  STRUCT
   S711A_WELD_DATA : STRUCT
    STATION_MAIN : WORD ;
    DISTINCTION_LH_RH : WORD ;
    STAION_NUMBER : WORD ;
    VIN_NUMBER1 : WORD ;
    VIN_NUMBER2 : WORD ;
    VIN_NUMBER3 : WORD ;
    VIN_NUMBER4 : WORD ;
    SEQ_NUMBER1 : WORD ;
    SEQ_NUMBER2 : WORD ;
    RBT1_BT_CODE_NO : WORD ;
    RBT1_WELD_COUNT : WORD ;
    RBT2_BT_CODE_NO : WORD ;
    RBT2_WELD_COUNT : WORD ;
    RBT3_BT_CODE_NO : WORD ;
    RBT3_WELD_COUNT : WORD ;
    RBT4_BT_CODE_NO : WORD ;
    RBT4_WELD_COUNT : WORD ;
    RBT5_BT_CODE_NO : WORD ;
    RBT5_WELD_COUNT : WORD ;
    RBT6_BT_CODE_NO : WORD ;
    RBT6_WELD_COUNT : WORD ;
    RBT7_BT_CODE_NO : WORD ;
    RBT7_WELD_COUNT : WORD ;
    RBT8_BT_CODE_NO : WORD ;
    RBT8_WELD_COUNT : WORD ;
    RBT9_BT_CODE_NO : WORD ;
    RBT9_WELD_COUNT : WORD ;
    RBT10_BT_CODE_NO : WORD ;
    RBT10_WELD_COUNT : WORD ;
    RBT11_BT_CODE_NO : WORD ;
    RBT11_WELD_COUNT : WORD ;
    RBT12_BT_CODE_NO : WORD ;
    RBT12_WELD_COUNT : WORD ;
    RBT13_BT_CODE_NO : WORD ;
    RBT13_WELD_COUNT : WORD ;
    RBT14_BT_CODE_NO : WORD ;
    RBT14_WELD_COUNT : WORD ;
    RBT15_BT_CODE_NO : WORD ;
    RBT15_WELD_COUNT : WORD ;
    RBT16_BT_CODE_NO : WORD ;
    RBT16_WELD_COUNT : WORD ;
    RBT17_BT_CODE_NO : WORD ;
    RBT17_WELD_COUNT : WORD ;
    RBT18_BT_CODE_NO : WORD ;
    RBT18_WELD_COUNT : WORD ;
    RBT19_BT_CODE_NO : WORD ;
    RBT19_WELD_COUNT : WORD ;
    RBT20_BT_CODE_NO : WORD ;
    RBT20_WELD_COUNT : WORD ;
    RBT21_BT_CODE_NO : WORD ;
    RBT21_WELD_COUNT : WORD ;
    RBT22_BT_CODE_NO : WORD ;
    RBT22_WELD_COUNT : WORD ;
    RBT23_BT_CODE_NO : WORD ;
    RBT23_WELD_COUNT : WORD ;
    RBT24_BT_CODE_NO : WORD ;
    RBT24_WELD_COUNT : WORD ;
    WELD_DETERMINES_RESULT : WORD ;
    WELD_CHECK_SUM : WORD ;
    SPARE1 : WORD ;
    SPARE2 : WORD ;
    SPARE3 : WORD ;
    SPARE4 : WORD ;
    SPARE5 : WORD ;
    SPARE6 : WORD ;
    SPARE7 : WORD ;
    SPARE8 : WORD ;
    SPARE9 : WORD ;
    SPARE10 : WORD ;
    SPARE11 : WORD ;
    SPARE12 : WORD ;
    SPARE13 : WORD ;
    SPARE14 : WORD ;
    SPARE15 : WORD ;
    SPARE16 : WORD ;
    SPARE17 : WORD ;
    SPARE18 : WORD ;
    SPARE19 : WORD ;
    SPARE20 : WORD ;
    SPARE21 : WORD ;
    SPARE22 : WORD ;
    SPARE23 : WORD ;
    SPARE24 : WORD ;
    SPARE25 : WORD ;
    SPARE26 : WORD ;
    SPARE27 : WORD ;
    SPARE28 : WORD ;
    SPARE29 : WORD ;
    SPARE30 : WORD ;
    SPARE31 : WORD ;
    RBT1_WELD_COUNT_OK : BOOL ;
    RBT1_WELD_COUNT_NG : BOOL ;
    RBT1_PASS_T_TAG : BOOL ;
    RBT1_PASS_L_TAG : BOOL ;
    RBT2_WELD_COUNT_OK : BOOL ;
    RBT2_WELD_COUNT_NG : BOOL ;
    RBT2_PASS_T_TAG : BOOL ;
    RBT2_PASS_L_TAG : BOOL ;
    RBT3_WELD_COUNT_OK : BOOL ;
    RBT3_WELD_COUNT_NG : BOOL ;
    RBT3_PASS_T_TAG : BOOL ;
    RBT3_PASS_L_TAG : BOOL ;
    RBT4_WELD_COUNT_OK : BOOL ;
    RBT4_WELD_COUNT_NG : BOOL ;
    RBT4_PASS_T_TAG : BOOL ;
    RBT4_PASS_L_TAG : BOOL ;
    RBT5_WELD_COUNT_OK : BOOL ;
    RBT5_WELD_COUNT_NG : BOOL ;
    RBT5_PASS_T_TAG : BOOL ;
    RBT5_PASS_L_TAG : BOOL ;
    RBT6_WELD_COUNT_OK : BOOL ;
    RBT6_WELD_COUNT_NG : BOOL ;
    RBT6_PASS_T_TAG : BOOL ;
    RBT6_PASS_L_TAG : BOOL ;
    RBT7_WELD_COUNT_OK : BOOL ;
    RBT7_WELD_COUNT_NG : BOOL ;
    RBT7_PASS_T_TAG : BOOL ;
    RBT7_PASS_L_TAG : BOOL ;
    RBT8_WELD_COUNT_OK : BOOL ;
    RBT8_WELD_COUNT_NG : BOOL ;
    RBT8_PASS_T_TAG : BOOL ;
    RBT8_PASS_L_TAG : BOOL ;
    RBT9_WELD_COUNT_OK : BOOL ;
    RBT9_WELD_COUNT_NG : BOOL ;
    RBT9_PASS_T_TAG : BOOL ;
    RBT9_PASS_L_TAG : BOOL ;
    RBT10_WELD_COUNT_OK : BOOL ;
    RBT10_WELD_COUNT_NG : BOOL ;
    RBT10_PASS_T_TAG : BOOL ;
    RBT10_PASS_L_TAG : BOOL ;
    RBT11_WELD_COUNT_OK : BOOL ;
    RBT11_WELD_COUNT_NG : BOOL ;
    RBT11_PASS_T_TAG : BOOL ;
    RBT11_PASS_L_TAG : BOOL ;
    RBT12_WELD_COUNT_OK : BOOL ;
    RBT12_WELD_COUNT_NG : BOOL ;
    RBT12_PASS_T_TAG : BOOL ;
    RBT12_PASS_L_TAG : BOOL ;
    RBT13_WELD_COUNT_OK : BOOL ;
    RBT13_WELD_COUNT_NG : BOOL ;
    RBT13_PASS_T_TAG : BOOL ;
    RBT13_PASS_L_TAG : BOOL ;
    RBT14_WELD_COUNT_OK : BOOL ;
    RBT14_WELD_COUNT_NG : BOOL ;
    RBT14_PASS_T_TAG : BOOL ;
    RBT14_PASS_L_TAG : BOOL ;
    RBT15_WELD_COUNT_OK : BOOL ;
    RBT15_WELD_COUNT_NG : BOOL ;
    RBT15_PASS_T_TAG : BOOL ;
    RBT15_PASS_L_TAG : BOOL ;
    RBT16_WELD_COUNT_OK : BOOL ;
    RBT16_WELD_COUNT_NG : BOOL ;
    RBT16_PASS_T_TAG : BOOL ;
    RBT16_PASS_L_TAG : BOOL ;
    RBT17_WELD_COUNT_OK : BOOL ;
    RBT17_WELD_COUNT_NG : BOOL ;
    RBT17_PASS_T_TAG : BOOL ;
    RBT17_PASS_L_TAG : BOOL ;
    RBT18_WELD_COUNT_OK : BOOL ;
    RBT18_WELD_COUNT_NG : BOOL ;
    RBT18_PASS_T_TAG : BOOL ;
    RBT18_PASS_L_TAG : BOOL ;
    RBT19_WELD_COUNT_OK : BOOL ;
    RBT19_WELD_COUNT_NG : BOOL ;
    RBT19_PASS_T_TAG : BOOL ;
    RBT19_PASS_L_TAG : BOOL ;
    RBT20_WELD_COUNT_OK : BOOL ;
    RBT20_WELD_COUNT_NG : BOOL ;
    RBT20_PASS_T_TAG : BOOL ;
    RBT20_PASS_L_TAG : BOOL ;
    RBT21_WELD_COUNT_OK : BOOL ;
    RBT21_WELD_COUNT_NG : BOOL ;
    RBT21_PASS_T_TAG : BOOL ;
    RBT21_PASS_L_TAG : BOOL ;
    RBT22_WELD_COUNT_OK : BOOL ;
    RBT22_WELD_COUNT_NG : BOOL ;
    RBT22_PASS_T_TAG : BOOL ;
    RBT22_PASS_L_TAG : BOOL ;
    RBT23_WELD_COUNT_OK : BOOL ;
    RBT23_WELD_COUNT_NG : BOOL ;
    RBT23_PASS_T_TAG : BOOL ;
    RBT23_PASS_L_TAG : BOOL ;
    RBT24_WELD_COUNT_OK : BOOL ;
    RBT24_WELD_COUNT_NG : BOOL ;
    RBT24_PASS_T_TAG : BOOL ;
    RBT24_PASS_L_TAG : BOOL ;
    SPARE100 : BOOL ;
    SPARE101 : BOOL ;
    SPARE102 : BOOL ;
    SPARE103 : BOOL ;
    SPARE104 : BOOL ;
    SPARE105 : BOOL ;
    SPARE106 : BOOL ;
    SPARE107 : BOOL ;
    SPARE108 : BOOL ;
    SPARE109 : BOOL ;
    SPARE110 : BOOL ;
    SPARE111 : BOOL ;
    SPARE112 : BOOL ;
    SPARE113 : BOOL ;
    SPARE114 : BOOL ;
    SPARE115 : BOOL ;
    SPARE116 : WORD ;
    SPARE117 : WORD ;
    SPARE118 : WORD ;
   END_STRUCT ;
   S706_WELD_DATA : STRUCT
    STATION_MAIN : WORD ;
    DISTINCTION_LH_RH : WORD ;
    STAION_NUMBER : WORD ;
    VIN_NUMBER1 : WORD ;
    VIN_NUMBER2 : WORD ;
    VIN_NUMBER3 : WORD ;
    VIN_NUMBER4 : WORD ;
    SEQ_NUMBER1 : WORD ;
    SEQ_NUMBER2 : WORD ;
    RBT1_BT_CODE_NO : WORD ;
    RBT1_WELD_COUNT : WORD ;
    RBT2_BT_CODE_NO : WORD ;
    RBT2_WELD_COUNT : WORD ;
    RBT3_BT_CODE_NO : WORD ;
    RBT3_WELD_COUNT : WORD ;
    RBT4_BT_CODE_NO : WORD ;
    RBT4_WELD_COUNT : WORD ;
    RBT5_BT_CODE_NO : WORD ;
    RBT5_WELD_COUNT : WORD ;
    RBT6_BT_CODE_NO : WORD ;
    RBT6_WELD_COUNT : WORD ;
    RBT7_BT_CODE_NO : WORD ;
    RBT7_WELD_COUNT : WORD ;
    RBT8_BT_CODE_NO : WORD ;
    RBT8_WELD_COUNT : WORD ;
    RBT9_BT_CODE_NO : WORD ;
    RBT9_WELD_COUNT : WORD ;
    RBT10_BT_CODE_NO : WORD ;
    RBT10_WELD_COUNT : WORD ;
    RBT11_BT_CODE_NO : WORD ;
    RBT11_WELD_COUNT : WORD ;
    RBT12_BT_CODE_NO : WORD ;
    RBT12_WELD_COUNT : WORD ;
    RBT13_BT_CODE_NO : WORD ;
    RBT13_WELD_COUNT : WORD ;
    RBT14_BT_CODE_NO : WORD ;
    RBT14_WELD_COUNT : WORD ;
    RBT15_BT_CODE_NO : WORD ;
    RBT15_WELD_COUNT : WORD ;
    RBT16_BT_CODE_NO : WORD ;
    RBT16_WELD_COUNT : WORD ;
    RBT17_BT_CODE_NO : WORD ;
    RBT17_WELD_COUNT : WORD ;
    RBT18_BT_CODE_NO : WORD ;
    RBT18_WELD_COUNT : WORD ;
    RBT19_BT_CODE_NO : WORD ;
    RBT19_WELD_COUNT : WORD ;
    RBT20_BT_CODE_NO : WORD ;
    RBT20_WELD_COUNT : WORD ;
    RBT21_BT_CODE_NO : WORD ;
    RBT21_WELD_COUNT : WORD ;
    RBT22_BT_CODE_NO : WORD ;
    RBT22_WELD_COUNT : WORD ;
    RBT23_BT_CODE_NO : WORD ;
    RBT23_WELD_COUNT : WORD ;
    RBT24_BT_CODE_NO : WORD ;
    RBT24_WELD_COUNT : WORD ;
    WELD_DETERMINES_RESULT : WORD ;
    WELD_CHECK_SUM : WORD ;
    SPARE1 : WORD ;
    SPARE2 : WORD ;
    SPARE3 : WORD ;
    SPARE4 : WORD ;
    SPARE5 : WORD ;
    SPARE6 : WORD ;
    SPARE7 : WORD ;
    SPARE8 : WORD ;
    SPARE9 : WORD ;
    SPARE10 : WORD ;
    SPARE11 : WORD ;
    SPARE12 : WORD ;
    SPARE13 : WORD ;
    SPARE14 : WORD ;
    SPARE15 : WORD ;
    SPARE16 : WORD ;
    SPARE17 : WORD ;
    SPARE18 : WORD ;
    SPARE19 : WORD ;
    SPARE20 : WORD ;
    SPARE21 : WORD ;
    SPARE22 : WORD ;
    SPARE23 : WORD ;
    SPARE24 : WORD ;
    SPARE25 : WORD ;
    SPARE26 : WORD ;
    SPARE27 : WORD ;
    SPARE28 : WORD ;
    SPARE29 : WORD ;
    SPARE30 : WORD ;
    SPARE31 : WORD ;
    RBT1_WELD_COUNT_OK : BOOL ;
    RBT1_WELD_COUNT_NG : BOOL ;
    RBT1_PASS_T_TAG : BOOL ;
    RBT1_PASS_L_TAG : BOOL ;
    RBT2_WELD_COUNT_OK : BOOL ;
    RBT2_WELD_COUNT_NG : BOOL ;
    RBT2_PASS_T_TAG : BOOL ;
    RBT2_PASS_L_TAG : BOOL ;
    RBT3_WELD_COUNT_OK : BOOL ;
    RBT3_WELD_COUNT_NG : BOOL ;
    RBT3_PASS_T_TAG : BOOL ;
    RBT3_PASS_L_TAG : BOOL ;
    RBT4_WELD_COUNT_OK : BOOL ;
    RBT4_WELD_COUNT_NG : BOOL ;
    RBT4_PASS_T_TAG : BOOL ;
    RBT4_PASS_L_TAG : BOOL ;
    RBT5_WELD_COUNT_OK : BOOL ;
    RBT5_WELD_COUNT_NG : BOOL ;
    RBT5_PASS_T_TAG : BOOL ;
    RBT5_PASS_L_TAG : BOOL ;
    RBT6_WELD_COUNT_OK : BOOL ;
    RBT6_WELD_COUNT_NG : BOOL ;
    RBT6_PASS_T_TAG : BOOL ;
    RBT6_PASS_L_TAG : BOOL ;
    RBT7_WELD_COUNT_OK : BOOL ;
    RBT7_WELD_COUNT_NG : BOOL ;
    RBT7_PASS_T_TAG : BOOL ;
    RBT7_PASS_L_TAG : BOOL ;
    RBT8_WELD_COUNT_OK : BOOL ;
    RBT8_WELD_COUNT_NG : BOOL ;
    RBT8_PASS_T_TAG : BOOL ;
    RBT8_PASS_L_TAG : BOOL ;
    RBT9_WELD_COUNT_OK : BOOL ;
    RBT9_WELD_COUNT_NG : BOOL ;
    RBT9_PASS_T_TAG : BOOL ;
    RBT9_PASS_L_TAG : BOOL ;
    RBT10_WELD_COUNT_OK : BOOL ;
    RBT10_WELD_COUNT_NG : BOOL ;
    RBT10_PASS_T_TAG : BOOL ;
    RBT10_PASS_L_TAG : BOOL ;
    RBT11_WELD_COUNT_OK : BOOL ;
    RBT11_WELD_COUNT_NG : BOOL ;
    RBT11_PASS_T_TAG : BOOL ;
    RBT11_PASS_L_TAG : BOOL ;
    RBT12_WELD_COUNT_OK : BOOL ;
    RBT12_WELD_COUNT_NG : BOOL ;
    RBT12_PASS_T_TAG : BOOL ;
    RBT12_PASS_L_TAG : BOOL ;
    RBT13_WELD_COUNT_OK : BOOL ;
    RBT13_WELD_COUNT_NG : BOOL ;
    RBT13_PASS_T_TAG : BOOL ;
    RBT13_PASS_L_TAG : BOOL ;
    RBT14_WELD_COUNT_OK : BOOL ;
    RBT14_WELD_COUNT_NG : BOOL ;
    RBT14_PASS_T_TAG : BOOL ;
    RBT14_PASS_L_TAG : BOOL ;
    RBT15_WELD_COUNT_OK : BOOL ;
    RBT15_WELD_COUNT_NG : BOOL ;
    RBT15_PASS_T_TAG : BOOL ;
    RBT15_PASS_L_TAG : BOOL ;
    RBT16_WELD_COUNT_OK : BOOL ;
    RBT16_WELD_COUNT_NG : BOOL ;
    RBT16_PASS_T_TAG : BOOL ;
    RBT16_PASS_L_TAG : BOOL ;
    RBT17_WELD_COUNT_OK : BOOL ;
    RBT17_WELD_COUNT_NG : BOOL ;
    RBT17_PASS_T_TAG : BOOL ;
    RBT17_PASS_L_TAG : BOOL ;
    RBT18_WELD_COUNT_OK : BOOL ;
    RBT18_WELD_COUNT_NG : BOOL ;
    RBT18_PASS_T_TAG : BOOL ;
    RBT18_PASS_L_TAG : BOOL ;
    RBT19_WELD_COUNT_OK : BOOL ;
    RBT19_WELD_COUNT_NG : BOOL ;
    RBT19_PASS_T_TAG : BOOL ;
    RBT19_PASS_L_TAG : BOOL ;
    RBT20_WELD_COUNT_OK : BOOL ;
    RBT20_WELD_COUNT_NG : BOOL ;
    RBT20_PASS_T_TAG : BOOL ;
    RBT20_PASS_L_TAG : BOOL ;
    RBT21_WELD_COUNT_OK : BOOL ;
    RBT21_WELD_COUNT_NG : BOOL ;
    RBT21_PASS_T_TAG : BOOL ;
    RBT21_PASS_L_TAG : BOOL ;
    RBT22_WELD_COUNT_OK : BOOL ;
    RBT22_WELD_COUNT_NG : BOOL ;
    RBT22_PASS_T_TAG : BOOL ;
    RBT22_PASS_L_TAG : BOOL ;
    RBT23_WELD_COUNT_OK : BOOL ;
    RBT23_WELD_COUNT_NG : BOOL ;
    RBT23_PASS_T_TAG : BOOL ;
    RBT23_PASS_L_TAG : BOOL ;
    RBT24_WELD_COUNT_OK : BOOL ;
    RBT24_WELD_COUNT_NG : BOOL ;
    RBT24_PASS_T_TAG : BOOL ;
    RBT24_PASS_L_TAG : BOOL ;
    SPARE100 : BOOL ;
    SPARE101 : BOOL ;
    SPARE102 : BOOL ;
    SPARE103 : BOOL ;
    SPARE104 : BOOL ;
    SPARE105 : BOOL ;
    SPARE106 : BOOL ;
    SPARE107 : BOOL ;
    SPARE108 : BOOL ;
    SPARE109 : BOOL ;
    SPARE110 : BOOL ;
    SPARE111 : BOOL ;
    SPARE112 : BOOL ;
    SPARE113 : BOOL ;
    SPARE114 : BOOL ;
    SPARE115 : BOOL ;
    SPARE116 : WORD ;
    SPARE117 : WORD ;
    SPARE118 : WORD ;
   END_STRUCT ;
   S711_WELD_DATA : STRUCT
    STATION_MAIN : WORD ;
    DISTINCTION_LH_RH : WORD ;
    STAION_NUMBER : WORD ;
    VIN_NUMBER1 : WORD ;
    VIN_NUMBER2 : WORD ;
    VIN_NUMBER3 : WORD ;
    VIN_NUMBER4 : WORD ;
    SEQ_NUMBER1 : WORD ;
    SEQ_NUMBER2 : WORD ;
    RBT1_BT_CODE_NO : WORD ;
    RBT1_WELD_COUNT : WORD ;
    RBT2_BT_CODE_NO : WORD ;
    RBT2_WELD_COUNT : WORD ;
    RBT3_BT_CODE_NO : WORD ;
    RBT3_WELD_COUNT : WORD ;
    RBT4_BT_CODE_NO : WORD ;
    RBT4_WELD_COUNT : WORD ;
    RBT5_BT_CODE_NO : WORD ;
    RBT5_WELD_COUNT : WORD ;
    RBT6_BT_CODE_NO : WORD ;
    RBT6_WELD_COUNT : WORD ;
    RBT7_BT_CODE_NO : WORD ;
    RBT7_WELD_COUNT : WORD ;
    RBT8_BT_CODE_NO : WORD ;
    RBT8_WELD_COUNT : WORD ;
    RBT9_BT_CODE_NO : WORD ;
    RBT9_WELD_COUNT : WORD ;
    RBT10_BT_CODE_NO : WORD ;
    RBT10_WELD_COUNT : WORD ;
    RBT11_BT_CODE_NO : WORD ;
    RBT11_WELD_COUNT : WORD ;
    RBT12_BT_CODE_NO : WORD ;
    RBT12_WELD_COUNT : WORD ;
    RBT13_BT_CODE_NO : WORD ;
    RBT13_WELD_COUNT : WORD ;
    RBT14_BT_CODE_NO : WORD ;
    RBT14_WELD_COUNT : WORD ;
    RBT15_BT_CODE_NO : WORD ;
    RBT15_WELD_COUNT : WORD ;
    RBT16_BT_CODE_NO : WORD ;
    RBT16_WELD_COUNT : WORD ;
    RBT17_BT_CODE_NO : WORD ;
    RBT17_WELD_COUNT : WORD ;
    RBT18_BT_CODE_NO : WORD ;
    RBT18_WELD_COUNT : WORD ;
    RBT19_BT_CODE_NO : WORD ;
    RBT19_WELD_COUNT : WORD ;
    RBT20_BT_CODE_NO : WORD ;
    RBT20_WELD_COUNT : WORD ;
    RBT21_BT_CODE_NO : WORD ;
    RBT21_WELD_COUNT : WORD ;
    RBT22_BT_CODE_NO : WORD ;
    RBT22_WELD_COUNT : WORD ;
    RBT23_BT_CODE_NO : WORD ;
    RBT23_WELD_COUNT : WORD ;
    RBT24_BT_CODE_NO : WORD ;
    RBT24_WELD_COUNT : WORD ;
    WELD_DETERMINES_RESULT : WORD ;
    WELD_CHECK_SUM : WORD ;
    SPARE1 : WORD ;
    SPARE2 : WORD ;
    SPARE3 : WORD ;
    SPARE4 : WORD ;
    SPARE5 : WORD ;
    SPARE6 : WORD ;
    SPARE7 : WORD ;
    SPARE8 : WORD ;
    SPARE9 : WORD ;
    SPARE10 : WORD ;
    SPARE11 : WORD ;
    SPARE12 : WORD ;
    SPARE13 : WORD ;
    SPARE14 : WORD ;
    SPARE15 : WORD ;
    SPARE16 : WORD ;
    SPARE17 : WORD ;
    SPARE18 : WORD ;
    SPARE19 : WORD ;
    SPARE20 : WORD ;
    SPARE21 : WORD ;
    SPARE22 : WORD ;
    SPARE23 : WORD ;
    SPARE24 : WORD ;
    SPARE25 : WORD ;
    SPARE26 : WORD ;
    SPARE27 : WORD ;
    SPARE28 : WORD ;
    SPARE29 : WORD ;
    SPARE30 : WORD ;
    SPARE31 : WORD ;
    RBT1_WELD_COUNT_OK : BOOL ;
    RBT1_WELD_COUNT_NG : BOOL ;
    RBT1_PASS_T_TAG : BOOL ;
    RBT1_PASS_L_TAG : BOOL ;
    RBT2_WELD_COUNT_OK : BOOL ;
    RBT2_WELD_COUNT_NG : BOOL ;
    RBT2_PASS_T_TAG : BOOL ;
    RBT2_PASS_L_TAG : BOOL ;
    RBT3_WELD_COUNT_OK : BOOL ;
    RBT3_WELD_COUNT_NG : BOOL ;
    RBT3_PASS_T_TAG : BOOL ;
    RBT3_PASS_L_TAG : BOOL ;
    RBT4_WELD_COUNT_OK : BOOL ;
    RBT4_WELD_COUNT_NG : BOOL ;
    RBT4_PASS_T_TAG : BOOL ;
    RBT4_PASS_L_TAG : BOOL ;
    RBT5_WELD_COUNT_OK : BOOL ;
    RBT5_WELD_COUNT_NG : BOOL ;
    RBT5_PASS_T_TAG : BOOL ;
    RBT5_PASS_L_TAG : BOOL ;
    RBT6_WELD_COUNT_OK : BOOL ;
    RBT6_WELD_COUNT_NG : BOOL ;
    RBT6_PASS_T_TAG : BOOL ;
    RBT6_PASS_L_TAG : BOOL ;
    RBT7_WELD_COUNT_OK : BOOL ;
    RBT7_WELD_COUNT_NG : BOOL ;
    RBT7_PASS_T_TAG : BOOL ;
    RBT7_PASS_L_TAG : BOOL ;
    RBT8_WELD_COUNT_OK : BOOL ;
    RBT8_WELD_COUNT_NG : BOOL ;
    RBT8_PASS_T_TAG : BOOL ;
    RBT8_PASS_L_TAG : BOOL ;
    RBT9_WELD_COUNT_OK : BOOL ;
    RBT9_WELD_COUNT_NG : BOOL ;
    RBT9_PASS_T_TAG : BOOL ;
    RBT9_PASS_L_TAG : BOOL ;
    RBT10_WELD_COUNT_OK : BOOL ;
    RBT10_WELD_COUNT_NG : BOOL ;
    RBT10_PASS_T_TAG : BOOL ;
    RBT10_PASS_L_TAG : BOOL ;
    RBT11_WELD_COUNT_OK : BOOL ;
    RBT11_WELD_COUNT_NG : BOOL ;
    RBT11_PASS_T_TAG : BOOL ;
    RBT11_PASS_L_TAG : BOOL ;
    RBT12_WELD_COUNT_OK : BOOL ;
    RBT12_WELD_COUNT_NG : BOOL ;
    RBT12_PASS_T_TAG : BOOL ;
    RBT12_PASS_L_TAG : BOOL ;
    RBT13_WELD_COUNT_OK : BOOL ;
    RBT13_WELD_COUNT_NG : BOOL ;
    RBT13_PASS_T_TAG : BOOL ;
    RBT13_PASS_L_TAG : BOOL ;
    RBT14_WELD_COUNT_OK : BOOL ;
    RBT14_WELD_COUNT_NG : BOOL ;
    RBT14_PASS_T_TAG : BOOL ;
    RBT14_PASS_L_TAG : BOOL ;
    RBT15_WELD_COUNT_OK : BOOL ;
    RBT15_WELD_COUNT_NG : BOOL ;
    RBT15_PASS_T_TAG : BOOL ;
    RBT15_PASS_L_TAG : BOOL ;
    RBT16_WELD_COUNT_OK : BOOL ;
    RBT16_WELD_COUNT_NG : BOOL ;
    RBT16_PASS_T_TAG : BOOL ;
    RBT16_PASS_L_TAG : BOOL ;
    RBT17_WELD_COUNT_OK : BOOL ;
    RBT17_WELD_COUNT_NG : BOOL ;
    RBT17_PASS_T_TAG : BOOL ;
    RBT17_PASS_L_TAG : BOOL ;
    RBT18_WELD_COUNT_OK : BOOL ;
    RBT18_WELD_COUNT_NG : BOOL ;
    RBT18_PASS_T_TAG : BOOL ;
    RBT18_PASS_L_TAG : BOOL ;
    RBT19_WELD_COUNT_OK : BOOL ;
    RBT19_WELD_COUNT_NG : BOOL ;
    RBT19_PASS_T_TAG : BOOL ;
    RBT19_PASS_L_TAG : BOOL ;
    RBT20_WELD_COUNT_OK : BOOL ;
    RBT20_WELD_COUNT_NG : BOOL ;
    RBT20_PASS_T_TAG : BOOL ;
    RBT20_PASS_L_TAG : BOOL ;
    RBT21_WELD_COUNT_OK : BOOL ;
    RBT21_WELD_COUNT_NG : BOOL ;
    RBT21_PASS_T_TAG : BOOL ;
    RBT21_PASS_L_TAG : BOOL ;
    RBT22_WELD_COUNT_OK : BOOL ;
    RBT22_WELD_COUNT_NG : BOOL ;
    RBT22_PASS_T_TAG : BOOL ;
    RBT22_PASS_L_TAG : BOOL ;
    RBT23_WELD_COUNT_OK : BOOL ;
    RBT23_WELD_COUNT_NG : BOOL ;
    RBT23_PASS_T_TAG : BOOL ;
    RBT23_PASS_L_TAG : BOOL ;
    RBT24_WELD_COUNT_OK : BOOL ;
    RBT24_WELD_COUNT_NG : BOOL ;
    RBT24_PASS_T_TAG : BOOL ;
    RBT24_PASS_L_TAG : BOOL ;
    SPARE100 : BOOL ;
    SPARE101 : BOOL ;
    SPARE102 : BOOL ;
    SPARE103 : BOOL ;
    SPARE104 : BOOL ;
    SPARE105 : BOOL ;
    SPARE106 : BOOL ;
    SPARE107 : BOOL ;
    SPARE108 : BOOL ;
    SPARE109 : BOOL ;
    SPARE110 : BOOL ;
    SPARE111 : BOOL ;
    SPARE112 : BOOL ;
    SPARE113 : BOOL ;
    SPARE114 : BOOL ;
    SPARE115 : BOOL ;
    SPARE116 : WORD ;
    SPARE117 : WORD ;
    SPARE118 : WORD ;
   END_STRUCT ;
  END_STRUCT ;
BEGIN
   S711A_WELD_DATA.STATION_MAIN := W#16#0;
   S711A_WELD_DATA.DISTINCTION_LH_RH := W#16#0;
   S711A_WELD_DATA.STAION_NUMBER := W#16#0;
   S711A_WELD_DATA.VIN_NUMBER1 := W#16#0;
   S711A_WELD_DATA.VIN_NUMBER2 := W#16#0;
   S711A_WELD_DATA.VIN_NUMBER3 := W#16#0;
   S711A_WELD_DATA.VIN_NUMBER4 := W#16#0;
   S711A_WELD_DATA.SEQ_NUMBER1 := W#16#0;
   S711A_WELD_DATA.SEQ_NUMBER2 := W#16#0;
   S711A_WELD_DATA.RBT1_BT_CODE_NO := W#16#0;
   S711A_WELD_DATA.RBT1_WELD_COUNT := W#16#0;
   S711A_WELD_DATA.RBT2_BT_CODE_NO := W#16#0;
   S711A_WELD_DATA.RBT2_WELD_COUNT := W#16#0;
   S711A_WELD_DATA.RBT3_BT_CODE_NO := W#16#0;
   S711A_WELD_DATA.RBT3_WELD_COUNT := W#16#0;
   S711A_WELD_DATA.RBT4_BT_CODE_NO := W#16#0;
   S711A_WELD_DATA.RBT4_WELD_COUNT := W#16#0;
   S711A_WELD_DATA.RBT5_BT_CODE_NO := W#16#0;
   S711A_WELD_DATA.RBT5_WELD_COUNT := W#16#0;
   S711A_WELD_DATA.RBT6_BT_CODE_NO := W#16#0;
   S711A_WELD_DATA.RBT6_WELD_COUNT := W#16#0;
   S711A_WELD_DATA.RBT7_BT_CODE_NO := W#16#0;
   S711A_WELD_DATA.RBT7_WELD_COUNT := W#16#0;
   S711A_WELD_DATA.RBT8_BT_CODE_NO := W#16#0;
   S711A_WELD_DATA.RBT8_WELD_COUNT := W#16#0;
   S711A_WELD_DATA.RBT9_BT_CODE_NO := W#16#0;
   S711A_WELD_DATA.RBT9_WELD_COUNT := W#16#0;
   S711A_WELD_DATA.RBT10_BT_CODE_NO := W#16#0;
   S711A_WELD_DATA.RBT10_WELD_COUNT := W#16#0;
   S711A_WELD_DATA.RBT11_BT_CODE_NO := W#16#0;
   S711A_WELD_DATA.RBT11_WELD_COUNT := W#16#0;
   S711A_WELD_DATA.RBT12_BT_CODE_NO := W#16#0;
   S711A_WELD_DATA.RBT12_WELD_COUNT := W#16#0;
   S711A_WELD_DATA.RBT13_BT_CODE_NO := W#16#0;
   S711A_WELD_DATA.RBT13_WELD_COUNT := W#16#0;
   S711A_WELD_DATA.RBT14_BT_CODE_NO := W#16#0;
   S711A_WELD_DATA.RBT14_WELD_COUNT := W#16#0;
   S711A_WELD_DATA.RBT15_BT_CODE_NO := W#16#0;
   S711A_WELD_DATA.RBT15_WELD_COUNT := W#16#0;
   S711A_WELD_DATA.RBT16_BT_CODE_NO := W#16#0;
   S711A_WELD_DATA.RBT16_WELD_COUNT := W#16#0;
   S711A_WELD_DATA.RBT17_BT_CODE_NO := W#16#0;
   S711A_WELD_DATA.RBT17_WELD_COUNT := W#16#0;
   S711A_WELD_DATA.RBT18_BT_CODE_NO := W#16#0;
   S711A_WELD_DATA.RBT18_WELD_COUNT := W#16#0;
   S711A_WELD_DATA.RBT19_BT_CODE_NO := W#16#0;
   S711A_WELD_DATA.RBT19_WELD_COUNT := W#16#0;
   S711A_WELD_DATA.RBT20_BT_CODE_NO := W#16#0;
   S711A_WELD_DATA.RBT20_WELD_COUNT := W#16#0;
   S711A_WELD_DATA.RBT21_BT_CODE_NO := W#16#0;
   S711A_WELD_DATA.RBT21_WELD_COUNT := W#16#0;
   S711A_WELD_DATA.RBT22_BT_CODE_NO := W#16#0;
   S711A_WELD_DATA.RBT22_WELD_COUNT := W#16#0;
   S711A_WELD_DATA.RBT23_BT_CODE_NO := W#16#0;
   S711A_WELD_DATA.RBT23_WELD_COUNT := W#16#0;
   S711A_WELD_DATA.RBT24_BT_CODE_NO := W#16#0;
   S711A_WELD_DATA.RBT24_WELD_COUNT := W#16#0;
   S711A_WELD_DATA.WELD_DETERMINES_RESULT := W#16#0;
   S711A_WELD_DATA.WELD_CHECK_SUM := W#16#0;
   S711A_WELD_DATA.SPARE1 := W#16#0;
   S711A_WELD_DATA.SPARE2 := W#16#0;
   S711A_WELD_DATA.SPARE3 := W#16#0;
   S711A_WELD_DATA.SPARE4 := W#16#0;
   S711A_WELD_DATA.SPARE5 := W#16#0;
   S711A_WELD_DATA.SPARE6 := W#16#0;
   S711A_WELD_DATA.SPARE7 := W#16#0;
   S711A_WELD_DATA.SPARE8 := W#16#0;
   S711A_WELD_DATA.SPARE9 := W#16#0;
   S711A_WELD_DATA.SPARE10 := W#16#0;
   S711A_WELD_DATA.SPARE11 := W#16#0;
   S711A_WELD_DATA.SPARE12 := W#16#0;
   S711A_WELD_DATA.SPARE13 := W#16#0;
   S711A_WELD_DATA.SPARE14 := W#16#0;
   S711A_WELD_DATA.SPARE15 := W#16#0;
   S711A_WELD_DATA.SPARE16 := W#16#0;
   S711A_WELD_DATA.SPARE17 := W#16#0;
   S711A_WELD_DATA.SPARE18 := W#16#0;
   S711A_WELD_DATA.SPARE19 := W#16#0;
   S711A_WELD_DATA.SPARE20 := W#16#0;
   S711A_WELD_DATA.SPARE21 := W#16#0;
   S711A_WELD_DATA.SPARE22 := W#16#0;
   S711A_WELD_DATA.SPARE23 := W#16#0;
   S711A_WELD_DATA.SPARE24 := W#16#0;
   S711A_WELD_DATA.SPARE25 := W#16#0;
   S711A_WELD_DATA.SPARE26 := W#16#0;
   S711A_WELD_DATA.SPARE27 := W#16#0;
   S711A_WELD_DATA.SPARE28 := W#16#0;
   S711A_WELD_DATA.SPARE29 := W#16#0;
   S711A_WELD_DATA.SPARE30 := W#16#0;
   S711A_WELD_DATA.SPARE31 := W#16#0;
   S711A_WELD_DATA.RBT1_WELD_COUNT_OK := FALSE;
   S711A_WELD_DATA.RBT1_WELD_COUNT_NG := FALSE;
   S711A_WELD_DATA.RBT1_PASS_T_TAG := FALSE;
   S711A_WELD_DATA.RBT1_PASS_L_TAG := FALSE;
   S711A_WELD_DATA.RBT2_WELD_COUNT_OK := FALSE;
   S711A_WELD_DATA.RBT2_WELD_COUNT_NG := FALSE;
   S711A_WELD_DATA.RBT2_PASS_T_TAG := FALSE;
   S711A_WELD_DATA.RBT2_PASS_L_TAG := FALSE;
   S711A_WELD_DATA.RBT3_WELD_COUNT_OK := FALSE;
   S711A_WELD_DATA.RBT3_WELD_COUNT_NG := FALSE;
   S711A_WELD_DATA.RBT3_PASS_T_TAG := FALSE;
   S711A_WELD_DATA.RBT3_PASS_L_TAG := FALSE;
   S711A_WELD_DATA.RBT4_WELD_COUNT_OK := FALSE;
   S711A_WELD_DATA.RBT4_WELD_COUNT_NG := FALSE;
   S711A_WELD_DATA.RBT4_PASS_T_TAG := FALSE;
   S711A_WELD_DATA.RBT4_PASS_L_TAG := FALSE;
   S711A_WELD_DATA.RBT5_WELD_COUNT_OK := FALSE;
   S711A_WELD_DATA.RBT5_WELD_COUNT_NG := FALSE;
   S711A_WELD_DATA.RBT5_PASS_T_TAG := FALSE;
   S711A_WELD_DATA.RBT5_PASS_L_TAG := FALSE;
   S711A_WELD_DATA.RBT6_WELD_COUNT_OK := FALSE;
   S711A_WELD_DATA.RBT6_WELD_COUNT_NG := FALSE;
   S711A_WELD_DATA.RBT6_PASS_T_TAG := FALSE;
   S711A_WELD_DATA.RBT6_PASS_L_TAG := FALSE;
   S711A_WELD_DATA.RBT7_WELD_COUNT_OK := FALSE;
   S711A_WELD_DATA.RBT7_WELD_COUNT_NG := FALSE;
   S711A_WELD_DATA.RBT7_PASS_T_TAG := FALSE;
   S711A_WELD_DATA.RBT7_PASS_L_TAG := FALSE;
   S711A_WELD_DATA.RBT8_WELD_COUNT_OK := FALSE;
   S711A_WELD_DATA.RBT8_WELD_COUNT_NG := FALSE;
   S711A_WELD_DATA.RBT8_PASS_T_TAG := FALSE;
   S711A_WELD_DATA.RBT8_PASS_L_TAG := FALSE;
   S711A_WELD_DATA.RBT9_WELD_COUNT_OK := FALSE;
   S711A_WELD_DATA.RBT9_WELD_COUNT_NG := FALSE;
   S711A_WELD_DATA.RBT9_PASS_T_TAG := FALSE;
   S711A_WELD_DATA.RBT9_PASS_L_TAG := FALSE;
   S711A_WELD_DATA.RBT10_WELD_COUNT_OK := FALSE;
   S711A_WELD_DATA.RBT10_WELD_COUNT_NG := FALSE;
   S711A_WELD_DATA.RBT10_PASS_T_TAG := FALSE;
   S711A_WELD_DATA.RBT10_PASS_L_TAG := FALSE;
   S711A_WELD_DATA.RBT11_WELD_COUNT_OK := FALSE;
   S711A_WELD_DATA.RBT11_WELD_COUNT_NG := FALSE;
   S711A_WELD_DATA.RBT11_PASS_T_TAG := FALSE;
   S711A_WELD_DATA.RBT11_PASS_L_TAG := FALSE;
   S711A_WELD_DATA.RBT12_WELD_COUNT_OK := FALSE;
   S711A_WELD_DATA.RBT12_WELD_COUNT_NG := FALSE;
   S711A_WELD_DATA.RBT12_PASS_T_TAG := FALSE;
   S711A_WELD_DATA.RBT12_PASS_L_TAG := FALSE;
   S711A_WELD_DATA.RBT13_WELD_COUNT_OK := FALSE;
   S711A_WELD_DATA.RBT13_WELD_COUNT_NG := FALSE;
   S711A_WELD_DATA.RBT13_PASS_T_TAG := FALSE;
   S711A_WELD_DATA.RBT13_PASS_L_TAG := FALSE;
   S711A_WELD_DATA.RBT14_WELD_COUNT_OK := FALSE;
   S711A_WELD_DATA.RBT14_WELD_COUNT_NG := FALSE;
   S711A_WELD_DATA.RBT14_PASS_T_TAG := FALSE;
   S711A_WELD_DATA.RBT14_PASS_L_TAG := FALSE;
   S711A_WELD_DATA.RBT15_WELD_COUNT_OK := FALSE;
   S711A_WELD_DATA.RBT15_WELD_COUNT_NG := FALSE;
   S711A_WELD_DATA.RBT15_PASS_T_TAG := FALSE;
   S711A_WELD_DATA.RBT15_PASS_L_TAG := FALSE;
   S711A_WELD_DATA.RBT16_WELD_COUNT_OK := FALSE;
   S711A_WELD_DATA.RBT16_WELD_COUNT_NG := FALSE;
   S711A_WELD_DATA.RBT16_PASS_T_TAG := FALSE;
   S711A_WELD_DATA.RBT16_PASS_L_TAG := FALSE;
   S711A_WELD_DATA.RBT17_WELD_COUNT_OK := FALSE;
   S711A_WELD_DATA.RBT17_WELD_COUNT_NG := FALSE;
   S711A_WELD_DATA.RBT17_PASS_T_TAG := FALSE;
   S711A_WELD_DATA.RBT17_PASS_L_TAG := FALSE;
   S711A_WELD_DATA.RBT18_WELD_COUNT_OK := FALSE;
   S711A_WELD_DATA.RBT18_WELD_COUNT_NG := FALSE;
   S711A_WELD_DATA.RBT18_PASS_T_TAG := FALSE;
   S711A_WELD_DATA.RBT18_PASS_L_TAG := FALSE;
   S711A_WELD_DATA.RBT19_WELD_COUNT_OK := FALSE;
   S711A_WELD_DATA.RBT19_WELD_COUNT_NG := FALSE;
   S711A_WELD_DATA.RBT19_PASS_T_TAG := FALSE;
   S711A_WELD_DATA.RBT19_PASS_L_TAG := FALSE;
   S711A_WELD_DATA.RBT20_WELD_COUNT_OK := FALSE;
   S711A_WELD_DATA.RBT20_WELD_COUNT_NG := FALSE;
   S711A_WELD_DATA.RBT20_PASS_T_TAG := FALSE;
   S711A_WELD_DATA.RBT20_PASS_L_TAG := FALSE;
   S711A_WELD_DATA.RBT21_WELD_COUNT_OK := FALSE;
   S711A_WELD_DATA.RBT21_WELD_COUNT_NG := FALSE;
   S711A_WELD_DATA.RBT21_PASS_T_TAG := FALSE;
   S711A_WELD_DATA.RBT21_PASS_L_TAG := FALSE;
   S711A_WELD_DATA.RBT22_WELD_COUNT_OK := FALSE;
   S711A_WELD_DATA.RBT22_WELD_COUNT_NG := FALSE;
   S711A_WELD_DATA.RBT22_PASS_T_TAG := FALSE;
   S711A_WELD_DATA.RBT22_PASS_L_TAG := FALSE;
   S711A_WELD_DATA.RBT23_WELD_COUNT_OK := FALSE;
   S711A_WELD_DATA.RBT23_WELD_COUNT_NG := FALSE;
   S711A_WELD_DATA.RBT23_PASS_T_TAG := FALSE;
   S711A_WELD_DATA.RBT23_PASS_L_TAG := FALSE;
   S711A_WELD_DATA.RBT24_WELD_COUNT_OK := FALSE;
   S711A_WELD_DATA.RBT24_WELD_COUNT_NG := FALSE;
   S711A_WELD_DATA.RBT24_PASS_T_TAG := FALSE;
   S711A_WELD_DATA.RBT24_PASS_L_TAG := FALSE;
   S711A_WELD_DATA.SPARE100 := FALSE;
   S711A_WELD_DATA.SPARE101 := FALSE;
   S711A_WELD_DATA.SPARE102 := FALSE;
   S711A_WELD_DATA.SPARE103 := FALSE;
   S711A_WELD_DATA.SPARE104 := FALSE;
   S711A_WELD_DATA.SPARE105 := FALSE;
   S711A_WELD_DATA.SPARE106 := FALSE;
   S711A_WELD_DATA.SPARE107 := FALSE;
   S711A_WELD_DATA.SPARE108 := FALSE;
   S711A_WELD_DATA.SPARE109 := FALSE;
   S711A_WELD_DATA.SPARE110 := FALSE;
   S711A_WELD_DATA.SPARE111 := FALSE;
   S711A_WELD_DATA.SPARE112 := FALSE;
   S711A_WELD_DATA.SPARE113 := FALSE;
   S711A_WELD_DATA.SPARE114 := FALSE;
   S711A_WELD_DATA.SPARE115 := FALSE;
   S711A_WELD_DATA.SPARE116 := W#16#0;
   S711A_WELD_DATA.SPARE117 := W#16#0;
   S711A_WELD_DATA.SPARE118 := W#16#0;
   S706_WELD_DATA.STATION_MAIN := W#16#0;
   S706_WELD_DATA.DISTINCTION_LH_RH := W#16#0;
   S706_WELD_DATA.STAION_NUMBER := W#16#0;
   S706_WELD_DATA.VIN_NUMBER1 := W#16#0;
   S706_WELD_DATA.VIN_NUMBER2 := W#16#0;
   S706_WELD_DATA.VIN_NUMBER3 := W#16#0;
   S706_WELD_DATA.VIN_NUMBER4 := W#16#0;
   S706_WELD_DATA.SEQ_NUMBER1 := W#16#0;
   S706_WELD_DATA.SEQ_NUMBER2 := W#16#0;
   S706_WELD_DATA.RBT1_BT_CODE_NO := W#16#0;
   S706_WELD_DATA.RBT1_WELD_COUNT := W#16#0;
   S706_WELD_DATA.RBT2_BT_CODE_NO := W#16#0;
   S706_WELD_DATA.RBT2_WELD_COUNT := W#16#0;
   S706_WELD_DATA.RBT3_BT_CODE_NO := W#16#0;
   S706_WELD_DATA.RBT3_WELD_COUNT := W#16#0;
   S706_WELD_DATA.RBT4_BT_CODE_NO := W#16#0;
   S706_WELD_DATA.RBT4_WELD_COUNT := W#16#0;
   S706_WELD_DATA.RBT5_BT_CODE_NO := W#16#0;
   S706_WELD_DATA.RBT5_WELD_COUNT := W#16#0;
   S706_WELD_DATA.RBT6_BT_CODE_NO := W#16#0;
   S706_WELD_DATA.RBT6_WELD_COUNT := W#16#0;
   S706_WELD_DATA.RBT7_BT_CODE_NO := W#16#0;
   S706_WELD_DATA.RBT7_WELD_COUNT := W#16#0;
   S706_WELD_DATA.RBT8_BT_CODE_NO := W#16#0;
   S706_WELD_DATA.RBT8_WELD_COUNT := W#16#0;
   S706_WELD_DATA.RBT9_BT_CODE_NO := W#16#0;
   S706_WELD_DATA.RBT9_WELD_COUNT := W#16#0;
   S706_WELD_DATA.RBT10_BT_CODE_NO := W#16#0;
   S706_WELD_DATA.RBT10_WELD_COUNT := W#16#0;
   S706_WELD_DATA.RBT11_BT_CODE_NO := W#16#0;
   S706_WELD_DATA.RBT11_WELD_COUNT := W#16#0;
   S706_WELD_DATA.RBT12_BT_CODE_NO := W#16#0;
   S706_WELD_DATA.RBT12_WELD_COUNT := W#16#0;
   S706_WELD_DATA.RBT13_BT_CODE_NO := W#16#0;
   S706_WELD_DATA.RBT13_WELD_COUNT := W#16#0;
   S706_WELD_DATA.RBT14_BT_CODE_NO := W#16#0;
   S706_WELD_DATA.RBT14_WELD_COUNT := W#16#0;
   S706_WELD_DATA.RBT15_BT_CODE_NO := W#16#0;
   S706_WELD_DATA.RBT15_WELD_COUNT := W#16#0;
   S706_WELD_DATA.RBT16_BT_CODE_NO := W#16#0;
   S706_WELD_DATA.RBT16_WELD_COUNT := W#16#0;
   S706_WELD_DATA.RBT17_BT_CODE_NO := W#16#0;
   S706_WELD_DATA.RBT17_WELD_COUNT := W#16#0;
   S706_WELD_DATA.RBT18_BT_CODE_NO := W#16#0;
   S706_WELD_DATA.RBT18_WELD_COUNT := W#16#0;
   S706_WELD_DATA.RBT19_BT_CODE_NO := W#16#0;
   S706_WELD_DATA.RBT19_WELD_COUNT := W#16#0;
   S706_WELD_DATA.RBT20_BT_CODE_NO := W#16#0;
   S706_WELD_DATA.RBT20_WELD_COUNT := W#16#0;
   S706_WELD_DATA.RBT21_BT_CODE_NO := W#16#0;
   S706_WELD_DATA.RBT21_WELD_COUNT := W#16#0;
   S706_WELD_DATA.RBT22_BT_CODE_NO := W#16#0;
   S706_WELD_DATA.RBT22_WELD_COUNT := W#16#0;
   S706_WELD_DATA.RBT23_BT_CODE_NO := W#16#0;
   S706_WELD_DATA.RBT23_WELD_COUNT := W#16#0;
   S706_WELD_DATA.RBT24_BT_CODE_NO := W#16#0;
   S706_WELD_DATA.RBT24_WELD_COUNT := W#16#0;
   S706_WELD_DATA.WELD_DETERMINES_RESULT := W#16#0;
   S706_WELD_DATA.WELD_CHECK_SUM := W#16#0;
   S706_WELD_DATA.SPARE1 := W#16#0;
   S706_WELD_DATA.SPARE2 := W#16#0;
   S706_WELD_DATA.SPARE3 := W#16#0;
   S706_WELD_DATA.SPARE4 := W#16#0;
   S706_WELD_DATA.SPARE5 := W#16#0;
   S706_WELD_DATA.SPARE6 := W#16#0;
   S706_WELD_DATA.SPARE7 := W#16#0;
   S706_WELD_DATA.SPARE8 := W#16#0;
   S706_WELD_DATA.SPARE9 := W#16#0;
   S706_WELD_DATA.SPARE10 := W#16#0;
   S706_WELD_DATA.SPARE11 := W#16#0;
   S706_WELD_DATA.SPARE12 := W#16#0;
   S706_WELD_DATA.SPARE13 := W#16#0;
   S706_WELD_DATA.SPARE14 := W#16#0;
   S706_WELD_DATA.SPARE15 := W#16#0;
   S706_WELD_DATA.SPARE16 := W#16#0;
   S706_WELD_DATA.SPARE17 := W#16#0;
   S706_WELD_DATA.SPARE18 := W#16#0;
   S706_WELD_DATA.SPARE19 := W#16#0;
   S706_WELD_DATA.SPARE20 := W#16#0;
   S706_WELD_DATA.SPARE21 := W#16#0;
   S706_WELD_DATA.SPARE22 := W#16#0;
   S706_WELD_DATA.SPARE23 := W#16#0;
   S706_WELD_DATA.SPARE24 := W#16#0;
   S706_WELD_DATA.SPARE25 := W#16#0;
   S706_WELD_DATA.SPARE26 := W#16#0;
   S706_WELD_DATA.SPARE27 := W#16#0;
   S706_WELD_DATA.SPARE28 := W#16#0;
   S706_WELD_DATA.SPARE29 := W#16#0;
   S706_WELD_DATA.SPARE30 := W#16#0;
   S706_WELD_DATA.SPARE31 := W#16#0;
   S706_WELD_DATA.RBT1_WELD_COUNT_OK := FALSE;
   S706_WELD_DATA.RBT1_WELD_COUNT_NG := FALSE;
   S706_WELD_DATA.RBT1_PASS_T_TAG := FALSE;
   S706_WELD_DATA.RBT1_PASS_L_TAG := FALSE;
   S706_WELD_DATA.RBT2_WELD_COUNT_OK := FALSE;
   S706_WELD_DATA.RBT2_WELD_COUNT_NG := FALSE;
   S706_WELD_DATA.RBT2_PASS_T_TAG := FALSE;
   S706_WELD_DATA.RBT2_PASS_L_TAG := FALSE;
   S706_WELD_DATA.RBT3_WELD_COUNT_OK := FALSE;
   S706_WELD_DATA.RBT3_WELD_COUNT_NG := FALSE;
   S706_WELD_DATA.RBT3_PASS_T_TAG := FALSE;
   S706_WELD_DATA.RBT3_PASS_L_TAG := FALSE;
   S706_WELD_DATA.RBT4_WELD_COUNT_OK := FALSE;
   S706_WELD_DATA.RBT4_WELD_COUNT_NG := FALSE;
   S706_WELD_DATA.RBT4_PASS_T_TAG := FALSE;
   S706_WELD_DATA.RBT4_PASS_L_TAG := FALSE;
   S706_WELD_DATA.RBT5_WELD_COUNT_OK := FALSE;
   S706_WELD_DATA.RBT5_WELD_COUNT_NG := FALSE;
   S706_WELD_DATA.RBT5_PASS_T_TAG := FALSE;
   S706_WELD_DATA.RBT5_PASS_L_TAG := FALSE;
   S706_WELD_DATA.RBT6_WELD_COUNT_OK := FALSE;
   S706_WELD_DATA.RBT6_WELD_COUNT_NG := FALSE;
   S706_WELD_DATA.RBT6_PASS_T_TAG := FALSE;
   S706_WELD_DATA.RBT6_PASS_L_TAG := FALSE;
   S706_WELD_DATA.RBT7_WELD_COUNT_OK := FALSE;
   S706_WELD_DATA.RBT7_WELD_COUNT_NG := FALSE;
   S706_WELD_DATA.RBT7_PASS_T_TAG := FALSE;
   S706_WELD_DATA.RBT7_PASS_L_TAG := FALSE;
   S706_WELD_DATA.RBT8_WELD_COUNT_OK := FALSE;
   S706_WELD_DATA.RBT8_WELD_COUNT_NG := FALSE;
   S706_WELD_DATA.RBT8_PASS_T_TAG := FALSE;
   S706_WELD_DATA.RBT8_PASS_L_TAG := FALSE;
   S706_WELD_DATA.RBT9_WELD_COUNT_OK := FALSE;
   S706_WELD_DATA.RBT9_WELD_COUNT_NG := FALSE;
   S706_WELD_DATA.RBT9_PASS_T_TAG := FALSE;
   S706_WELD_DATA.RBT9_PASS_L_TAG := FALSE;
   S706_WELD_DATA.RBT10_WELD_COUNT_OK := FALSE;
   S706_WELD_DATA.RBT10_WELD_COUNT_NG := FALSE;
   S706_WELD_DATA.RBT10_PASS_T_TAG := FALSE;
   S706_WELD_DATA.RBT10_PASS_L_TAG := FALSE;
   S706_WELD_DATA.RBT11_WELD_COUNT_OK := FALSE;
   S706_WELD_DATA.RBT11_WELD_COUNT_NG := FALSE;
   S706_WELD_DATA.RBT11_PASS_T_TAG := FALSE;
   S706_WELD_DATA.RBT11_PASS_L_TAG := FALSE;
   S706_WELD_DATA.RBT12_WELD_COUNT_OK := FALSE;
   S706_WELD_DATA.RBT12_WELD_COUNT_NG := FALSE;
   S706_WELD_DATA.RBT12_PASS_T_TAG := FALSE;
   S706_WELD_DATA.RBT12_PASS_L_TAG := FALSE;
   S706_WELD_DATA.RBT13_WELD_COUNT_OK := FALSE;
   S706_WELD_DATA.RBT13_WELD_COUNT_NG := FALSE;
   S706_WELD_DATA.RBT13_PASS_T_TAG := FALSE;
   S706_WELD_DATA.RBT13_PASS_L_TAG := FALSE;
   S706_WELD_DATA.RBT14_WELD_COUNT_OK := FALSE;
   S706_WELD_DATA.RBT14_WELD_COUNT_NG := FALSE;
   S706_WELD_DATA.RBT14_PASS_T_TAG := FALSE;
   S706_WELD_DATA.RBT14_PASS_L_TAG := FALSE;
   S706_WELD_DATA.RBT15_WELD_COUNT_OK := FALSE;
   S706_WELD_DATA.RBT15_WELD_COUNT_NG := FALSE;
   S706_WELD_DATA.RBT15_PASS_T_TAG := FALSE;
   S706_WELD_DATA.RBT15_PASS_L_TAG := FALSE;
   S706_WELD_DATA.RBT16_WELD_COUNT_OK := FALSE;
   S706_WELD_DATA.RBT16_WELD_COUNT_NG := FALSE;
   S706_WELD_DATA.RBT16_PASS_T_TAG := FALSE;
   S706_WELD_DATA.RBT16_PASS_L_TAG := FALSE;
   S706_WELD_DATA.RBT17_WELD_COUNT_OK := FALSE;
   S706_WELD_DATA.RBT17_WELD_COUNT_NG := FALSE;
   S706_WELD_DATA.RBT17_PASS_T_TAG := FALSE;
   S706_WELD_DATA.RBT17_PASS_L_TAG := FALSE;
   S706_WELD_DATA.RBT18_WELD_COUNT_OK := FALSE;
   S706_WELD_DATA.RBT18_WELD_COUNT_NG := FALSE;
   S706_WELD_DATA.RBT18_PASS_T_TAG := FALSE;
   S706_WELD_DATA.RBT18_PASS_L_TAG := FALSE;
   S706_WELD_DATA.RBT19_WELD_COUNT_OK := FALSE;
   S706_WELD_DATA.RBT19_WELD_COUNT_NG := FALSE;
   S706_WELD_DATA.RBT19_PASS_T_TAG := FALSE;
   S706_WELD_DATA.RBT19_PASS_L_TAG := FALSE;
   S706_WELD_DATA.RBT20_WELD_COUNT_OK := FALSE;
   S706_WELD_DATA.RBT20_WELD_COUNT_NG := FALSE;
   S706_WELD_DATA.RBT20_PASS_T_TAG := FALSE;
   S706_WELD_DATA.RBT20_PASS_L_TAG := FALSE;
   S706_WELD_DATA.RBT21_WELD_COUNT_OK := FALSE;
   S706_WELD_DATA.RBT21_WELD_COUNT_NG := FALSE;
   S706_WELD_DATA.RBT21_PASS_T_TAG := FALSE;
   S706_WELD_DATA.RBT21_PASS_L_TAG := FALSE;
   S706_WELD_DATA.RBT22_WELD_COUNT_OK := FALSE;
   S706_WELD_DATA.RBT22_WELD_COUNT_NG := FALSE;
   S706_WELD_DATA.RBT22_PASS_T_TAG := FALSE;
   S706_WELD_DATA.RBT22_PASS_L_TAG := FALSE;
   S706_WELD_DATA.RBT23_WELD_COUNT_OK := FALSE;
   S706_WELD_DATA.RBT23_WELD_COUNT_NG := FALSE;
   S706_WELD_DATA.RBT23_PASS_T_TAG := FALSE;
   S706_WELD_DATA.RBT23_PASS_L_TAG := FALSE;
   S706_WELD_DATA.RBT24_WELD_COUNT_OK := FALSE;
   S706_WELD_DATA.RBT24_WELD_COUNT_NG := FALSE;
   S706_WELD_DATA.RBT24_PASS_T_TAG := FALSE;
   S706_WELD_DATA.RBT24_PASS_L_TAG := FALSE;
   S706_WELD_DATA.SPARE100 := FALSE;
   S706_WELD_DATA.SPARE101 := FALSE;
   S706_WELD_DATA.SPARE102 := FALSE;
   S706_WELD_DATA.SPARE103 := FALSE;
   S706_WELD_DATA.SPARE104 := FALSE;
   S706_WELD_DATA.SPARE105 := FALSE;
   S706_WELD_DATA.SPARE106 := FALSE;
   S706_WELD_DATA.SPARE107 := FALSE;
   S706_WELD_DATA.SPARE108 := FALSE;
   S706_WELD_DATA.SPARE109 := FALSE;
   S706_WELD_DATA.SPARE110 := FALSE;
   S706_WELD_DATA.SPARE111 := FALSE;
   S706_WELD_DATA.SPARE112 := FALSE;
   S706_WELD_DATA.SPARE113 := FALSE;
   S706_WELD_DATA.SPARE114 := FALSE;
   S706_WELD_DATA.SPARE115 := FALSE;
   S706_WELD_DATA.SPARE116 := W#16#0;
   S706_WELD_DATA.SPARE117 := W#16#0;
   S706_WELD_DATA.SPARE118 := W#16#0;
   S711_WELD_DATA.STATION_MAIN := W#16#0;
   S711_WELD_DATA.DISTINCTION_LH_RH := W#16#0;
   S711_WELD_DATA.STAION_NUMBER := W#16#0;
   S711_WELD_DATA.VIN_NUMBER1 := W#16#0;
   S711_WELD_DATA.VIN_NUMBER2 := W#16#0;
   S711_WELD_DATA.VIN_NUMBER3 := W#16#0;
   S711_WELD_DATA.VIN_NUMBER4 := W#16#0;
   S711_WELD_DATA.SEQ_NUMBER1 := W#16#0;
   S711_WELD_DATA.SEQ_NUMBER2 := W#16#0;
   S711_WELD_DATA.RBT1_BT_CODE_NO := W#16#0;
   S711_WELD_DATA.RBT1_WELD_COUNT := W#16#0;
   S711_WELD_DATA.RBT2_BT_CODE_NO := W#16#0;
   S711_WELD_DATA.RBT2_WELD_COUNT := W#16#0;
   S711_WELD_DATA.RBT3_BT_CODE_NO := W#16#0;
   S711_WELD_DATA.RBT3_WELD_COUNT := W#16#0;
   S711_WELD_DATA.RBT4_BT_CODE_NO := W#16#0;
   S711_WELD_DATA.RBT4_WELD_COUNT := W#16#0;
   S711_WELD_DATA.RBT5_BT_CODE_NO := W#16#0;
   S711_WELD_DATA.RBT5_WELD_COUNT := W#16#0;
   S711_WELD_DATA.RBT6_BT_CODE_NO := W#16#0;
   S711_WELD_DATA.RBT6_WELD_COUNT := W#16#0;
   S711_WELD_DATA.RBT7_BT_CODE_NO := W#16#0;
   S711_WELD_DATA.RBT7_WELD_COUNT := W#16#0;
   S711_WELD_DATA.RBT8_BT_CODE_NO := W#16#0;
   S711_WELD_DATA.RBT8_WELD_COUNT := W#16#0;
   S711_WELD_DATA.RBT9_BT_CODE_NO := W#16#0;
   S711_WELD_DATA.RBT9_WELD_COUNT := W#16#0;
   S711_WELD_DATA.RBT10_BT_CODE_NO := W#16#0;
   S711_WELD_DATA.RBT10_WELD_COUNT := W#16#0;
   S711_WELD_DATA.RBT11_BT_CODE_NO := W#16#0;
   S711_WELD_DATA.RBT11_WELD_COUNT := W#16#0;
   S711_WELD_DATA.RBT12_BT_CODE_NO := W#16#0;
   S711_WELD_DATA.RBT12_WELD_COUNT := W#16#0;
   S711_WELD_DATA.RBT13_BT_CODE_NO := W#16#0;
   S711_WELD_DATA.RBT13_WELD_COUNT := W#16#0;
   S711_WELD_DATA.RBT14_BT_CODE_NO := W#16#0;
   S711_WELD_DATA.RBT14_WELD_COUNT := W#16#0;
   S711_WELD_DATA.RBT15_BT_CODE_NO := W#16#0;
   S711_WELD_DATA.RBT15_WELD_COUNT := W#16#0;
   S711_WELD_DATA.RBT16_BT_CODE_NO := W#16#0;
   S711_WELD_DATA.RBT16_WELD_COUNT := W#16#0;
   S711_WELD_DATA.RBT17_BT_CODE_NO := W#16#0;
   S711_WELD_DATA.RBT17_WELD_COUNT := W#16#0;
   S711_WELD_DATA.RBT18_BT_CODE_NO := W#16#0;
   S711_WELD_DATA.RBT18_WELD_COUNT := W#16#0;
   S711_WELD_DATA.RBT19_BT_CODE_NO := W#16#0;
   S711_WELD_DATA.RBT19_WELD_COUNT := W#16#0;
   S711_WELD_DATA.RBT20_BT_CODE_NO := W#16#0;
   S711_WELD_DATA.RBT20_WELD_COUNT := W#16#0;
   S711_WELD_DATA.RBT21_BT_CODE_NO := W#16#0;
   S711_WELD_DATA.RBT21_WELD_COUNT := W#16#0;
   S711_WELD_DATA.RBT22_BT_CODE_NO := W#16#0;
   S711_WELD_DATA.RBT22_WELD_COUNT := W#16#0;
   S711_WELD_DATA.RBT23_BT_CODE_NO := W#16#0;
   S711_WELD_DATA.RBT23_WELD_COUNT := W#16#0;
   S711_WELD_DATA.RBT24_BT_CODE_NO := W#16#0;
   S711_WELD_DATA.RBT24_WELD_COUNT := W#16#0;
   S711_WELD_DATA.WELD_DETERMINES_RESULT := W#16#0;
   S711_WELD_DATA.WELD_CHECK_SUM := W#16#0;
   S711_WELD_DATA.SPARE1 := W#16#0;
   S711_WELD_DATA.SPARE2 := W#16#0;
   S711_WELD_DATA.SPARE3 := W#16#0;
   S711_WELD_DATA.SPARE4 := W#16#0;
   S711_WELD_DATA.SPARE5 := W#16#0;
   S711_WELD_DATA.SPARE6 := W#16#0;
   S711_WELD_DATA.SPARE7 := W#16#0;
   S711_WELD_DATA.SPARE8 := W#16#0;
   S711_WELD_DATA.SPARE9 := W#16#0;
   S711_WELD_DATA.SPARE10 := W#16#0;
   S711_WELD_DATA.SPARE11 := W#16#0;
   S711_WELD_DATA.SPARE12 := W#16#0;
   S711_WELD_DATA.SPARE13 := W#16#0;
   S711_WELD_DATA.SPARE14 := W#16#0;
   S711_WELD_DATA.SPARE15 := W#16#0;
   S711_WELD_DATA.SPARE16 := W#16#0;
   S711_WELD_DATA.SPARE17 := W#16#0;
   S711_WELD_DATA.SPARE18 := W#16#0;
   S711_WELD_DATA.SPARE19 := W#16#0;
   S711_WELD_DATA.SPARE20 := W#16#0;
   S711_WELD_DATA.SPARE21 := W#16#0;
   S711_WELD_DATA.SPARE22 := W#16#0;
   S711_WELD_DATA.SPARE23 := W#16#0;
   S711_WELD_DATA.SPARE24 := W#16#0;
   S711_WELD_DATA.SPARE25 := W#16#0;
   S711_WELD_DATA.SPARE26 := W#16#0;
   S711_WELD_DATA.SPARE27 := W#16#0;
   S711_WELD_DATA.SPARE28 := W#16#0;
   S711_WELD_DATA.SPARE29 := W#16#0;
   S711_WELD_DATA.SPARE30 := W#16#0;
   S711_WELD_DATA.SPARE31 := W#16#0;
   S711_WELD_DATA.RBT1_WELD_COUNT_OK := FALSE;
   S711_WELD_DATA.RBT1_WELD_COUNT_NG := FALSE;
   S711_WELD_DATA.RBT1_PASS_T_TAG := FALSE;
   S711_WELD_DATA.RBT1_PASS_L_TAG := FALSE;
   S711_WELD_DATA.RBT2_WELD_COUNT_OK := FALSE;
   S711_WELD_DATA.RBT2_WELD_COUNT_NG := FALSE;
   S711_WELD_DATA.RBT2_PASS_T_TAG := FALSE;
   S711_WELD_DATA.RBT2_PASS_L_TAG := FALSE;
   S711_WELD_DATA.RBT3_WELD_COUNT_OK := FALSE;
   S711_WELD_DATA.RBT3_WELD_COUNT_NG := FALSE;
   S711_WELD_DATA.RBT3_PASS_T_TAG := FALSE;
   S711_WELD_DATA.RBT3_PASS_L_TAG := FALSE;
   S711_WELD_DATA.RBT4_WELD_COUNT_OK := FALSE;
   S711_WELD_DATA.RBT4_WELD_COUNT_NG := FALSE;
   S711_WELD_DATA.RBT4_PASS_T_TAG := FALSE;
   S711_WELD_DATA.RBT4_PASS_L_TAG := FALSE;
   S711_WELD_DATA.RBT5_WELD_COUNT_OK := FALSE;
   S711_WELD_DATA.RBT5_WELD_COUNT_NG := FALSE;
   S711_WELD_DATA.RBT5_PASS_T_TAG := FALSE;
   S711_WELD_DATA.RBT5_PASS_L_TAG := FALSE;
   S711_WELD_DATA.RBT6_WELD_COUNT_OK := FALSE;
   S711_WELD_DATA.RBT6_WELD_COUNT_NG := FALSE;
   S711_WELD_DATA.RBT6_PASS_T_TAG := FALSE;
   S711_WELD_DATA.RBT6_PASS_L_TAG := FALSE;
   S711_WELD_DATA.RBT7_WELD_COUNT_OK := FALSE;
   S711_WELD_DATA.RBT7_WELD_COUNT_NG := FALSE;
   S711_WELD_DATA.RBT7_PASS_T_TAG := FALSE;
   S711_WELD_DATA.RBT7_PASS_L_TAG := FALSE;
   S711_WELD_DATA.RBT8_WELD_COUNT_OK := FALSE;
   S711_WELD_DATA.RBT8_WELD_COUNT_NG := FALSE;
   S711_WELD_DATA.RBT8_PASS_T_TAG := FALSE;
   S711_WELD_DATA.RBT8_PASS_L_TAG := FALSE;
   S711_WELD_DATA.RBT9_WELD_COUNT_OK := FALSE;
   S711_WELD_DATA.RBT9_WELD_COUNT_NG := FALSE;
   S711_WELD_DATA.RBT9_PASS_T_TAG := FALSE;
   S711_WELD_DATA.RBT9_PASS_L_TAG := FALSE;
   S711_WELD_DATA.RBT10_WELD_COUNT_OK := FALSE;
   S711_WELD_DATA.RBT10_WELD_COUNT_NG := FALSE;
   S711_WELD_DATA.RBT10_PASS_T_TAG := FALSE;
   S711_WELD_DATA.RBT10_PASS_L_TAG := FALSE;
   S711_WELD_DATA.RBT11_WELD_COUNT_OK := FALSE;
   S711_WELD_DATA.RBT11_WELD_COUNT_NG := FALSE;
   S711_WELD_DATA.RBT11_PASS_T_TAG := FALSE;
   S711_WELD_DATA.RBT11_PASS_L_TAG := FALSE;
   S711_WELD_DATA.RBT12_WELD_COUNT_OK := FALSE;
   S711_WELD_DATA.RBT12_WELD_COUNT_NG := FALSE;
   S711_WELD_DATA.RBT12_PASS_T_TAG := FALSE;
   S711_WELD_DATA.RBT12_PASS_L_TAG := FALSE;
   S711_WELD_DATA.RBT13_WELD_COUNT_OK := FALSE;
   S711_WELD_DATA.RBT13_WELD_COUNT_NG := FALSE;
   S711_WELD_DATA.RBT13_PASS_T_TAG := FALSE;
   S711_WELD_DATA.RBT13_PASS_L_TAG := FALSE;
   S711_WELD_DATA.RBT14_WELD_COUNT_OK := FALSE;
   S711_WELD_DATA.RBT14_WELD_COUNT_NG := FALSE;
   S711_WELD_DATA.RBT14_PASS_T_TAG := FALSE;
   S711_WELD_DATA.RBT14_PASS_L_TAG := FALSE;
   S711_WELD_DATA.RBT15_WELD_COUNT_OK := FALSE;
   S711_WELD_DATA.RBT15_WELD_COUNT_NG := FALSE;
   S711_WELD_DATA.RBT15_PASS_T_TAG := FALSE;
   S711_WELD_DATA.RBT15_PASS_L_TAG := FALSE;
   S711_WELD_DATA.RBT16_WELD_COUNT_OK := FALSE;
   S711_WELD_DATA.RBT16_WELD_COUNT_NG := FALSE;
   S711_WELD_DATA.RBT16_PASS_T_TAG := FALSE;
   S711_WELD_DATA.RBT16_PASS_L_TAG := FALSE;
   S711_WELD_DATA.RBT17_WELD_COUNT_OK := FALSE;
   S711_WELD_DATA.RBT17_WELD_COUNT_NG := FALSE;
   S711_WELD_DATA.RBT17_PASS_T_TAG := FALSE;
   S711_WELD_DATA.RBT17_PASS_L_TAG := FALSE;
   S711_WELD_DATA.RBT18_WELD_COUNT_OK := FALSE;
   S711_WELD_DATA.RBT18_WELD_COUNT_NG := FALSE;
   S711_WELD_DATA.RBT18_PASS_T_TAG := FALSE;
   S711_WELD_DATA.RBT18_PASS_L_TAG := FALSE;
   S711_WELD_DATA.RBT19_WELD_COUNT_OK := FALSE;
   S711_WELD_DATA.RBT19_WELD_COUNT_NG := FALSE;
   S711_WELD_DATA.RBT19_PASS_T_TAG := FALSE;
   S711_WELD_DATA.RBT19_PASS_L_TAG := FALSE;
   S711_WELD_DATA.RBT20_WELD_COUNT_OK := FALSE;
   S711_WELD_DATA.RBT20_WELD_COUNT_NG := FALSE;
   S711_WELD_DATA.RBT20_PASS_T_TAG := FALSE;
   S711_WELD_DATA.RBT20_PASS_L_TAG := FALSE;
   S711_WELD_DATA.RBT21_WELD_COUNT_OK := FALSE;
   S711_WELD_DATA.RBT21_WELD_COUNT_NG := FALSE;
   S711_WELD_DATA.RBT21_PASS_T_TAG := FALSE;
   S711_WELD_DATA.RBT21_PASS_L_TAG := FALSE;
   S711_WELD_DATA.RBT22_WELD_COUNT_OK := FALSE;
   S711_WELD_DATA.RBT22_WELD_COUNT_NG := FALSE;
   S711_WELD_DATA.RBT22_PASS_T_TAG := FALSE;
   S711_WELD_DATA.RBT22_PASS_L_TAG := FALSE;
   S711_WELD_DATA.RBT23_WELD_COUNT_OK := FALSE;
   S711_WELD_DATA.RBT23_WELD_COUNT_NG := FALSE;
   S711_WELD_DATA.RBT23_PASS_T_TAG := FALSE;
   S711_WELD_DATA.RBT23_PASS_L_TAG := FALSE;
   S711_WELD_DATA.RBT24_WELD_COUNT_OK := FALSE;
   S711_WELD_DATA.RBT24_WELD_COUNT_NG := FALSE;
   S711_WELD_DATA.RBT24_PASS_T_TAG := FALSE;
   S711_WELD_DATA.RBT24_PASS_L_TAG := FALSE;
   S711_WELD_DATA.SPARE100 := FALSE;
   S711_WELD_DATA.SPARE101 := FALSE;
   S711_WELD_DATA.SPARE102 := FALSE;
   S711_WELD_DATA.SPARE103 := FALSE;
   S711_WELD_DATA.SPARE104 := FALSE;
   S711_WELD_DATA.SPARE105 := FALSE;
   S711_WELD_DATA.SPARE106 := FALSE;
   S711_WELD_DATA.SPARE107 := FALSE;
   S711_WELD_DATA.SPARE108 := FALSE;
   S711_WELD_DATA.SPARE109 := FALSE;
   S711_WELD_DATA.SPARE110 := FALSE;
   S711_WELD_DATA.SPARE111 := FALSE;
   S711_WELD_DATA.SPARE112 := FALSE;
   S711_WELD_DATA.SPARE113 := FALSE;
   S711_WELD_DATA.SPARE114 := FALSE;
   S711_WELD_DATA.SPARE115 := FALSE;
   S711_WELD_DATA.SPARE116 := W#16#0;
   S711_WELD_DATA.SPARE117 := W#16#0;
   S711_WELD_DATA.SPARE118 := W#16#0;
END_DATA_BLOCK

DATA_BLOCK DB 43
TITLE =
VERSION : 0.1


  STRUCT
   S711A_WELD_BUFF_DATA1 : STRUCT
    STATION_MAIN : WORD ;
    DISTINCTION_LH_RH : WORD ;
    STAION_NUMBER : WORD ;
    VIN_NUMBER1 : WORD ;
    VIN_NUMBER2 : WORD ;
    VIN_NUMBER3 : WORD ;
    VIN_NUMBER4 : WORD ;
    SEQ_NUMBER1 : WORD ;
    SEQ_NUMBER2 : WORD ;
    RBT1_BT_CODE_NO : WORD ;
    RBT1_WELD_COUNT : WORD ;
    RBT2_BT_CODE_NO : WORD ;
    RBT2_WELD_COUNT : WORD ;
    RBT3_BT_CODE_NO : WORD ;
    RBT3_WELD_COUNT : WORD ;
    RBT4_BT_CODE_NO : WORD ;
    RBT4_WELD_COUNT : WORD ;
    RBT5_BT_CODE_NO : WORD ;
    RBT5_WELD_COUNT : WORD ;
    RBT6_BT_CODE_NO : WORD ;
    RBT6_WELD_COUNT : WORD ;
    RBT7_BT_CODE_NO : WORD ;
    RBT7_WELD_COUNT : WORD ;
    RBT8_BT_CODE_NO : WORD ;
    RBT8_WELD_COUNT : WORD ;
    RBT9_BT_CODE_NO : WORD ;
    RBT9_WELD_COUNT : WORD ;
    RBT10_BT_CODE_NO : WORD ;
    RBT10_WELD_COUNT : WORD ;
    RBT11_BT_CODE_NO : WORD ;
    RBT11_WELD_COUNT : WORD ;
    RBT12_BT_CODE_NO : WORD ;
    RBT12_WELD_COUNT : WORD ;
    RBT13_BT_CODE_NO : WORD ;
    RBT13_WELD_COUNT : WORD ;
    RBT14_BT_CODE_NO : WORD ;
    RBT14_WELD_COUNT : WORD ;
    RBT15_BT_CODE_NO : WORD ;
    RBT15_WELD_COUNT : WORD ;
    RBT16_BT_CODE_NO : WORD ;
    RBT16_WELD_COUNT : WORD ;
    RBT17_BT_CODE_NO : WORD ;
    RBT17_WELD_COUNT : WORD ;
    RBT18_BT_CODE_NO : WORD ;
    RBT18_WELD_COUNT : WORD ;
    RBT19_BT_CODE_NO : WORD ;
    RBT19_WELD_COUNT : WORD ;
    RBT20_BT_CODE_NO : WORD ;
    RBT20_WELD_COUNT : WORD ;
    RBT21_BT_CODE_NO : WORD ;
    RBT21_WELD_COUNT : WORD ;
    RBT22_BT_CODE_NO : WORD ;
    RBT22_WELD_COUNT : WORD ;
    RBT23_BT_CODE_NO : WORD ;
    RBT23_WELD_COUNT : WORD ;
    RBT24_BT_CODE_NO : WORD ;
    RBT24_WELD_COUNT : WORD ;
    WELD_DETERMINES_RESULT : WORD ;
    WELD_CHECK_SUM : WORD ;
    SPARE1 : WORD ;
   END_STRUCT ;
   S711A_WELD_BUFF_DATA2 : STRUCT
    STATION_MAIN : WORD ;
    DISTINCTION_LH_RH : WORD ;
    STAION_NUMBER : WORD ;
    VIN_NUMBER1 : WORD ;
    VIN_NUMBER2 : WORD ;
    VIN_NUMBER3 : WORD ;
    VIN_NUMBER4 : WORD ;
    SEQ_NUMBER1 : WORD ;
    SEQ_NUMBER2 : WORD ;
    RBT1_BT_CODE_NO : WORD ;
    RBT1_WELD_COUNT : WORD ;
    RBT2_BT_CODE_NO : WORD ;
    RBT2_WELD_COUNT : WORD ;
    RBT3_BT_CODE_NO : WORD ;
    RBT3_WELD_COUNT : WORD ;
    RBT4_BT_CODE_NO : WORD ;
    RBT4_WELD_COUNT : WORD ;
    RBT5_BT_CODE_NO : WORD ;
    RBT5_WELD_COUNT : WORD ;
    RBT6_BT_CODE_NO : WORD ;
    RBT6_WELD_COUNT : WORD ;
    RBT7_BT_CODE_NO : WORD ;
    RBT7_WELD_COUNT : WORD ;
    RBT8_BT_CODE_NO : WORD ;
    RBT8_WELD_COUNT : WORD ;
    RBT9_BT_CODE_NO : WORD ;
    RBT9_WELD_COUNT : WORD ;
    RBT10_BT_CODE_NO : WORD ;
    RBT10_WELD_COUNT : WORD ;
    RBT11_BT_CODE_NO : WORD ;
    RBT11_WELD_COUNT : WORD ;
    RBT12_BT_CODE_NO : WORD ;
    RBT12_WELD_COUNT : WORD ;
    RBT13_BT_CODE_NO : WORD ;
    RBT13_WELD_COUNT : WORD ;
    RBT14_BT_CODE_NO : WORD ;
    RBT14_WELD_COUNT : WORD ;
    RBT15_BT_CODE_NO : WORD ;
    RBT15_WELD_COUNT : WORD ;
    RBT16_BT_CODE_NO : WORD ;
    RBT16_WELD_COUNT : WORD ;
    RBT17_BT_CODE_NO : WORD ;
    RBT17_WELD_COUNT : WORD ;
    RBT18_BT_CODE_NO : WORD ;
    RBT18_WELD_COUNT : WORD ;
    RBT19_BT_CODE_NO : WORD ;
    RBT19_WELD_COUNT : WORD ;
    RBT20_BT_CODE_NO : WORD ;
    RBT20_WELD_COUNT : WORD ;
    RBT21_BT_CODE_NO : WORD ;
    RBT21_WELD_COUNT : WORD ;
    RBT22_BT_CODE_NO : WORD ;
    RBT22_WELD_COUNT : WORD ;
    RBT23_BT_CODE_NO : WORD ;
    RBT23_WELD_COUNT : WORD ;
    RBT24_BT_CODE_NO : WORD ;
    RBT24_WELD_COUNT : WORD ;
    WELD_DETERMINES_RESULT : WORD ;
    WELD_CHECK_SUM : WORD ;
    SPARE1 : WORD ;
   END_STRUCT ;
   S711A_WELD_BUFF_DATA3 : STRUCT
    STATION_MAIN : WORD ;
    DISTINCTION_LH_RH : WORD ;
    STAION_NUMBER : WORD ;
    VIN_NUMBER1 : WORD ;
    VIN_NUMBER2 : WORD ;
    VIN_NUMBER3 : WORD ;
    VIN_NUMBER4 : WORD ;
    SEQ_NUMBER1 : WORD ;
    SEQ_NUMBER2 : WORD ;
    RBT1_BT_CODE_NO : WORD ;
    RBT1_WELD_COUNT : WORD ;
    RBT2_BT_CODE_NO : WORD ;
    RBT2_WELD_COUNT : WORD ;
    RBT3_BT_CODE_NO : WORD ;
    RBT3_WELD_COUNT : WORD ;
    RBT4_BT_CODE_NO : WORD ;
    RBT4_WELD_COUNT : WORD ;
    RBT5_BT_CODE_NO : WORD ;
    RBT5_WELD_COUNT : WORD ;
    RBT6_BT_CODE_NO : WORD ;
    RBT6_WELD_COUNT : WORD ;
    RBT7_BT_CODE_NO : WORD ;
    RBT7_WELD_COUNT : WORD ;
    RBT8_BT_CODE_NO : WORD ;
    RBT8_WELD_COUNT : WORD ;
    RBT9_BT_CODE_NO : WORD ;
    RBT9_WELD_COUNT : WORD ;
    RBT10_BT_CODE_NO : WORD ;
    RBT10_WELD_COUNT : WORD ;
    RBT11_BT_CODE_NO : WORD ;
    RBT11_WELD_COUNT : WORD ;
    RBT12_BT_CODE_NO : WORD ;
    RBT12_WELD_COUNT : WORD ;
    RBT13_BT_CODE_NO : WORD ;
    RBT13_WELD_COUNT : WORD ;
    RBT14_BT_CODE_NO : WORD ;
    RBT14_WELD_COUNT : WORD ;
    RBT15_BT_CODE_NO : WORD ;
    RBT15_WELD_COUNT : WORD ;
    RBT16_BT_CODE_NO : WORD ;
    RBT16_WELD_COUNT : WORD ;
    RBT17_BT_CODE_NO : WORD ;
    RBT17_WELD_COUNT : WORD ;
    RBT18_BT_CODE_NO : WORD ;
    RBT18_WELD_COUNT : WORD ;
    RBT19_BT_CODE_NO : WORD ;
    RBT19_WELD_COUNT : WORD ;
    RBT20_BT_CODE_NO : WORD ;
    RBT20_WELD_COUNT : WORD ;
    RBT21_BT_CODE_NO : WORD ;
    RBT21_WELD_COUNT : WORD ;
    RBT22_BT_CODE_NO : WORD ;
    RBT22_WELD_COUNT : WORD ;
    RBT23_BT_CODE_NO : WORD ;
    RBT23_WELD_COUNT : WORD ;
    RBT24_BT_CODE_NO : WORD ;
    RBT24_WELD_COUNT : WORD ;
    WELD_DETERMINES_RESULT : WORD ;
    WELD_CHECK_SUM : WORD ;
    SPARE1 : WORD ;
   END_STRUCT ;
   S711A_WELD_BUFF_DATA4 : STRUCT
    STATION_MAIN : WORD ;
    DISTINCTION_LH_RH : WORD ;
    STAION_NUMBER : WORD ;
    VIN_NUMBER1 : WORD ;
    VIN_NUMBER2 : WORD ;
    VIN_NUMBER3 : WORD ;
    VIN_NUMBER4 : WORD ;
    SEQ_NUMBER1 : WORD ;
    SEQ_NUMBER2 : WORD ;
    RBT1_BT_CODE_NO : WORD ;
    RBT1_WELD_COUNT : WORD ;
    RBT2_BT_CODE_NO : WORD ;
    RBT2_WELD_COUNT : WORD ;
    RBT3_BT_CODE_NO : WORD ;
    RBT3_WELD_COUNT : WORD ;
    RBT4_BT_CODE_NO : WORD ;
    RBT4_WELD_COUNT : WORD ;
    RBT5_BT_CODE_NO : WORD ;
    RBT5_WELD_COUNT : WORD ;
    RBT6_BT_CODE_NO : WORD ;
    RBT6_WELD_COUNT : WORD ;
    RBT7_BT_CODE_NO : WORD ;
    RBT7_WELD_COUNT : WORD ;
    RBT8_BT_CODE_NO : WORD ;
    RBT8_WELD_COUNT : WORD ;
    RBT9_BT_CODE_NO : WORD ;
    RBT9_WELD_COUNT : WORD ;
    RBT10_BT_CODE_NO : WORD ;
    RBT10_WELD_COUNT : WORD ;
    RBT11_BT_CODE_NO : WORD ;
    RBT11_WELD_COUNT : WORD ;
    RBT12_BT_CODE_NO : WORD ;
    RBT12_WELD_COUNT : WORD ;
    RBT13_BT_CODE_NO : WORD ;
    RBT13_WELD_COUNT : WORD ;
    RBT14_BT_CODE_NO : WORD ;
    RBT14_WELD_COUNT : WORD ;
    RBT15_BT_CODE_NO : WORD ;
    RBT15_WELD_COUNT : WORD ;
    RBT16_BT_CODE_NO : WORD ;
    RBT16_WELD_COUNT : WORD ;
    RBT17_BT_CODE_NO : WORD ;
    RBT17_WELD_COUNT : WORD ;
    RBT18_BT_CODE_NO : WORD ;
    RBT18_WELD_COUNT : WORD ;
    RBT19_BT_CODE_NO : WORD ;
    RBT19_WELD_COUNT : WORD ;
    RBT20_BT_CODE_NO : WORD ;
    RBT20_WELD_COUNT : WORD ;
    RBT21_BT_CODE_NO : WORD ;
    RBT21_WELD_COUNT : WORD ;
    RBT22_BT_CODE_NO : WORD ;
    RBT22_WELD_COUNT : WORD ;
    RBT23_BT_CODE_NO : WORD ;
    RBT23_WELD_COUNT : WORD ;
    RBT24_BT_CODE_NO : WORD ;
    RBT24_WELD_COUNT : WORD ;
    WELD_DETERMINES_RESULT : WORD ;
    WELD_CHECK_SUM : WORD ;
    SPARE1 : WORD ;
   END_STRUCT ;
   S711A_WELD_BUFF_DATA5 : STRUCT
    STATION_MAIN : WORD ;
    DISTINCTION_LH_RH : WORD ;
    STAION_NUMBER : WORD ;
    VIN_NUMBER1 : WORD ;
    VIN_NUMBER2 : WORD ;
    VIN_NUMBER3 : WORD ;
    VIN_NUMBER4 : WORD ;
    SEQ_NUMBER1 : WORD ;
    SEQ_NUMBER2 : WORD ;
    RBT1_BT_CODE_NO : WORD ;
    RBT1_WELD_COUNT : WORD ;
    RBT2_BT_CODE_NO : WORD ;
    RBT2_WELD_COUNT : WORD ;
    RBT3_BT_CODE_NO : WORD ;
    RBT3_WELD_COUNT : WORD ;
    RBT4_BT_CODE_NO : WORD ;
    RBT4_WELD_COUNT : WORD ;
    RBT5_BT_CODE_NO : WORD ;
    RBT5_WELD_COUNT : WORD ;
    RBT6_BT_CODE_NO : WORD ;
    RBT6_WELD_COUNT : WORD ;
    RBT7_BT_CODE_NO : WORD ;
    RBT7_WELD_COUNT : WORD ;
    RBT8_BT_CODE_NO : WORD ;
    RBT8_WELD_COUNT : WORD ;
    RBT9_BT_CODE_NO : WORD ;
    RBT9_WELD_COUNT : WORD ;
    RBT10_BT_CODE_NO : WORD ;
    RBT10_WELD_COUNT : WORD ;
    RBT11_BT_CODE_NO : WORD ;
    RBT11_WELD_COUNT : WORD ;
    RBT12_BT_CODE_NO : WORD ;
    RBT12_WELD_COUNT : WORD ;
    RBT13_BT_CODE_NO : WORD ;
    RBT13_WELD_COUNT : WORD ;
    RBT14_BT_CODE_NO : WORD ;
    RBT14_WELD_COUNT : WORD ;
    RBT15_BT_CODE_NO : WORD ;
    RBT15_WELD_COUNT : WORD ;
    RBT16_BT_CODE_NO : WORD ;
    RBT16_WELD_COUNT : WORD ;
    RBT17_BT_CODE_NO : WORD ;
    RBT17_WELD_COUNT : WORD ;
    RBT18_BT_CODE_NO : WORD ;
    RBT18_WELD_COUNT : WORD ;
    RBT19_BT_CODE_NO : WORD ;
    RBT19_WELD_COUNT : WORD ;
    RBT20_BT_CODE_NO : WORD ;
    RBT20_WELD_COUNT : WORD ;
    RBT21_BT_CODE_NO : WORD ;
    RBT21_WELD_COUNT : WORD ;
    RBT22_BT_CODE_NO : WORD ;
    RBT22_WELD_COUNT : WORD ;
    RBT23_BT_CODE_NO : WORD ;
    RBT23_WELD_COUNT : WORD ;
    RBT24_BT_CODE_NO : WORD ;
    RBT24_WELD_COUNT : WORD ;
    WELD_DETERMINES_RESULT : WORD ;
    WELD_CHECK_SUM : WORD ;
    SPARE1 : WORD ;
   END_STRUCT ;
   S711A_WELD_BUFF_DATA6 : STRUCT
    STATION_MAIN : WORD ;
    DISTINCTION_LH_RH : WORD ;
    STAION_NUMBER : WORD ;
    VIN_NUMBER1 : WORD ;
    VIN_NUMBER2 : WORD ;
    VIN_NUMBER3 : WORD ;
    VIN_NUMBER4 : WORD ;
    SEQ_NUMBER1 : WORD ;
    SEQ_NUMBER2 : WORD ;
    RBT1_BT_CODE_NO : WORD ;
    RBT1_WELD_COUNT : WORD ;
    RBT2_BT_CODE_NO : WORD ;
    RBT2_WELD_COUNT : WORD ;
    RBT3_BT_CODE_NO : WORD ;
    RBT3_WELD_COUNT : WORD ;
    RBT4_BT_CODE_NO : WORD ;
    RBT4_WELD_COUNT : WORD ;
    RBT5_BT_CODE_NO : WORD ;
    RBT5_WELD_COUNT : WORD ;
    RBT6_BT_CODE_NO : WORD ;
    RBT6_WELD_COUNT : WORD ;
    RBT7_BT_CODE_NO : WORD ;
    RBT7_WELD_COUNT : WORD ;
    RBT8_BT_CODE_NO : WORD ;
    RBT8_WELD_COUNT : WORD ;
    RBT9_BT_CODE_NO : WORD ;
    RBT9_WELD_COUNT : WORD ;
    RBT10_BT_CODE_NO : WORD ;
    RBT10_WELD_COUNT : WORD ;
    RBT11_BT_CODE_NO : WORD ;
    RBT11_WELD_COUNT : WORD ;
    RBT12_BT_CODE_NO : WORD ;
    RBT12_WELD_COUNT : WORD ;
    RBT13_BT_CODE_NO : WORD ;
    RBT13_WELD_COUNT : WORD ;
    RBT14_BT_CODE_NO : WORD ;
    RBT14_WELD_COUNT : WORD ;
    RBT15_BT_CODE_NO : WORD ;
    RBT15_WELD_COUNT : WORD ;
    RBT16_BT_CODE_NO : WORD ;
    RBT16_WELD_COUNT : WORD ;
    RBT17_BT_CODE_NO : WORD ;
    RBT17_WELD_COUNT : WORD ;
    RBT18_BT_CODE_NO : WORD ;
    RBT18_WELD_COUNT : WORD ;
    RBT19_BT_CODE_NO : WORD ;
    RBT19_WELD_COUNT : WORD ;
    RBT20_BT_CODE_NO : WORD ;
    RBT20_WELD_COUNT : WORD ;
    RBT21_BT_CODE_NO : WORD ;
    RBT21_WELD_COUNT : WORD ;
    RBT22_BT_CODE_NO : WORD ;
    RBT22_WELD_COUNT : WORD ;
    RBT23_BT_CODE_NO : WORD ;
    RBT23_WELD_COUNT : WORD ;
    RBT24_BT_CODE_NO : WORD ;
    RBT24_WELD_COUNT : WORD ;
    WELD_DETERMINES_RESULT : WORD ;
    WELD_CHECK_SUM : WORD ;
    SPARE1 : WORD ;
   END_STRUCT ;
   S711A_WELD_BUFF_DATA7 : STRUCT
    STATION_MAIN : WORD ;
    DISTINCTION_LH_RH : WORD ;
    STAION_NUMBER : WORD ;
    VIN_NUMBER1 : WORD ;
    VIN_NUMBER2 : WORD ;
    VIN_NUMBER3 : WORD ;
    VIN_NUMBER4 : WORD ;
    SEQ_NUMBER1 : WORD ;
    SEQ_NUMBER2 : WORD ;
    RBT1_BT_CODE_NO : WORD ;
    RBT1_WELD_COUNT : WORD ;
    RBT2_BT_CODE_NO : WORD ;
    RBT2_WELD_COUNT : WORD ;
    RBT3_BT_CODE_NO : WORD ;
    RBT3_WELD_COUNT : WORD ;
    RBT4_BT_CODE_NO : WORD ;
    RBT4_WELD_COUNT : WORD ;
    RBT5_BT_CODE_NO : WORD ;
    RBT5_WELD_COUNT : WORD ;
    RBT6_BT_CODE_NO : WORD ;
    RBT6_WELD_COUNT : WORD ;
    RBT7_BT_CODE_NO : WORD ;
    RBT7_WELD_COUNT : WORD ;
    RBT8_BT_CODE_NO : WORD ;
    RBT8_WELD_COUNT : WORD ;
    RBT9_BT_CODE_NO : WORD ;
    RBT9_WELD_COUNT : WORD ;
    RBT10_BT_CODE_NO : WORD ;
    RBT10_WELD_COUNT : WORD ;
    RBT11_BT_CODE_NO : WORD ;
    RBT11_WELD_COUNT : WORD ;
    RBT12_BT_CODE_NO : WORD ;
    RBT12_WELD_COUNT : WORD ;
    RBT13_BT_CODE_NO : WORD ;
    RBT13_WELD_COUNT : WORD ;
    RBT14_BT_CODE_NO : WORD ;
    RBT14_WELD_COUNT : WORD ;
    RBT15_BT_CODE_NO : WORD ;
    RBT15_WELD_COUNT : WORD ;
    RBT16_BT_CODE_NO : WORD ;
    RBT16_WELD_COUNT : WORD ;
    RBT17_BT_CODE_NO : WORD ;
    RBT17_WELD_COUNT : WORD ;
    RBT18_BT_CODE_NO : WORD ;
    RBT18_WELD_COUNT : WORD ;
    RBT19_BT_CODE_NO : WORD ;
    RBT19_WELD_COUNT : WORD ;
    RBT20_BT_CODE_NO : WORD ;
    RBT20_WELD_COUNT : WORD ;
    RBT21_BT_CODE_NO : WORD ;
    RBT21_WELD_COUNT : WORD ;
    RBT22_BT_CODE_NO : WORD ;
    RBT22_WELD_COUNT : WORD ;
    RBT23_BT_CODE_NO : WORD ;
    RBT23_WELD_COUNT : WORD ;
    RBT24_BT_CODE_NO : WORD ;
    RBT24_WELD_COUNT : WORD ;
    WELD_DETERMINES_RESULT : WORD ;
    WELD_CHECK_SUM : WORD ;
    SPARE1 : WORD ;
   END_STRUCT ;
   S711A_WELD_BUFF_DATA8 : STRUCT
    STATION_MAIN : WORD ;
    DISTINCTION_LH_RH : WORD ;
    STAION_NUMBER : WORD ;
    VIN_NUMBER1 : WORD ;
    VIN_NUMBER2 : WORD ;
    VIN_NUMBER3 : WORD ;
    VIN_NUMBER4 : WORD ;
    SEQ_NUMBER1 : WORD ;
    SEQ_NUMBER2 : WORD ;
    RBT1_BT_CODE_NO : WORD ;
    RBT1_WELD_COUNT : WORD ;
    RBT2_BT_CODE_NO : WORD ;
    RBT2_WELD_COUNT : WORD ;
    RBT3_BT_CODE_NO : WORD ;
    RBT3_WELD_COUNT : WORD ;
    RBT4_BT_CODE_NO : WORD ;
    RBT4_WELD_COUNT : WORD ;
    RBT5_BT_CODE_NO : WORD ;
    RBT5_WELD_COUNT : WORD ;
    RBT6_BT_CODE_NO : WORD ;
    RBT6_WELD_COUNT : WORD ;
    RBT7_BT_CODE_NO : WORD ;
    RBT7_WELD_COUNT : WORD ;
    RBT8_BT_CODE_NO : WORD ;
    RBT8_WELD_COUNT : WORD ;
    RBT9_BT_CODE_NO : WORD ;
    RBT9_WELD_COUNT : WORD ;
    RBT10_BT_CODE_NO : WORD ;
    RBT10_WELD_COUNT : WORD ;
    RBT11_BT_CODE_NO : WORD ;
    RBT11_WELD_COUNT : WORD ;
    RBT12_BT_CODE_NO : WORD ;
    RBT12_WELD_COUNT : WORD ;
    RBT13_BT_CODE_NO : WORD ;
    RBT13_WELD_COUNT : WORD ;
    RBT14_BT_CODE_NO : WORD ;
    RBT14_WELD_COUNT : WORD ;
    RBT15_BT_CODE_NO : WORD ;
    RBT15_WELD_COUNT : WORD ;
    RBT16_BT_CODE_NO : WORD ;
    RBT16_WELD_COUNT : WORD ;
    RBT17_BT_CODE_NO : WORD ;
    RBT17_WELD_COUNT : WORD ;
    RBT18_BT_CODE_NO : WORD ;
    RBT18_WELD_COUNT : WORD ;
    RBT19_BT_CODE_NO : WORD ;
    RBT19_WELD_COUNT : WORD ;
    RBT20_BT_CODE_NO : WORD ;
    RBT20_WELD_COUNT : WORD ;
    RBT21_BT_CODE_NO : WORD ;
    RBT21_WELD_COUNT : WORD ;
    RBT22_BT_CODE_NO : WORD ;
    RBT22_WELD_COUNT : WORD ;
    RBT23_BT_CODE_NO : WORD ;
    RBT23_WELD_COUNT : WORD ;
    RBT24_BT_CODE_NO : WORD ;
    RBT24_WELD_COUNT : WORD ;
    WELD_DETERMINES_RESULT : WORD ;
    WELD_CHECK_SUM : WORD ;
    SPARE1 : WORD ;
   END_STRUCT ;
   S711A_WELD_BUFF_DATA9 : STRUCT
    STATION_MAIN : WORD ;
    DISTINCTION_LH_RH : WORD ;
    STAION_NUMBER : WORD ;
    VIN_NUMBER1 : WORD ;
    VIN_NUMBER2 : WORD ;
    VIN_NUMBER3 : WORD ;
    VIN_NUMBER4 : WORD ;
    SEQ_NUMBER1 : WORD ;
    SEQ_NUMBER2 : WORD ;
    RBT1_BT_CODE_NO : WORD ;
    RBT1_WELD_COUNT : WORD ;
    RBT2_BT_CODE_NO : WORD ;
    RBT2_WELD_COUNT : WORD ;
    RBT3_BT_CODE_NO : WORD ;
    RBT3_WELD_COUNT : WORD ;
    RBT4_BT_CODE_NO : WORD ;
    RBT4_WELD_COUNT : WORD ;
    RBT5_BT_CODE_NO : WORD ;
    RBT5_WELD_COUNT : WORD ;
    RBT6_BT_CODE_NO : WORD ;
    RBT6_WELD_COUNT : WORD ;
    RBT7_BT_CODE_NO : WORD ;
    RBT7_WELD_COUNT : WORD ;
    RBT8_BT_CODE_NO : WORD ;
    RBT8_WELD_COUNT : WORD ;
    RBT9_BT_CODE_NO : WORD ;
    RBT9_WELD_COUNT : WORD ;
    RBT10_BT_CODE_NO : WORD ;
    RBT10_WELD_COUNT : WORD ;
    RBT11_BT_CODE_NO : WORD ;
    RBT11_WELD_COUNT : WORD ;
    RBT12_BT_CODE_NO : WORD ;
    RBT12_WELD_COUNT : WORD ;
    RBT13_BT_CODE_NO : WORD ;
    RBT13_WELD_COUNT : WORD ;
    RBT14_BT_CODE_NO : WORD ;
    RBT14_WELD_COUNT : WORD ;
    RBT15_BT_CODE_NO : WORD ;
    RBT15_WELD_COUNT : WORD ;
    RBT16_BT_CODE_NO : WORD ;
    RBT16_WELD_COUNT : WORD ;
    RBT17_BT_CODE_NO : WORD ;
    RBT17_WELD_COUNT : WORD ;
    RBT18_BT_CODE_NO : WORD ;
    RBT18_WELD_COUNT : WORD ;
    RBT19_BT_CODE_NO : WORD ;
    RBT19_WELD_COUNT : WORD ;
    RBT20_BT_CODE_NO : WORD ;
    RBT20_WELD_COUNT : WORD ;
    RBT21_BT_CODE_NO : WORD ;
    RBT21_WELD_COUNT : WORD ;
    RBT22_BT_CODE_NO : WORD ;
    RBT22_WELD_COUNT : WORD ;
    RBT23_BT_CODE_NO : WORD ;
    RBT23_WELD_COUNT : WORD ;
    RBT24_BT_CODE_NO : WORD ;
    RBT24_WELD_COUNT : WORD ;
    WELD_DETERMINES_RESULT : WORD ;
    WELD_CHECK_SUM : WORD ;
    SPARE1 : WORD ;
   END_STRUCT ;
   S711A_WELD_BUFF_DATA10 : STRUCT
    STATION_MAIN : WORD ;
    DISTINCTION_LH_RH : WORD ;
    STAION_NUMBER : WORD ;
    VIN_NUMBER1 : WORD ;
    VIN_NUMBER2 : WORD ;
    VIN_NUMBER3 : WORD ;
    VIN_NUMBER4 : WORD ;
    SEQ_NUMBER1 : WORD ;
    SEQ_NUMBER2 : WORD ;
    RBT1_BT_CODE_NO : WORD ;
    RBT1_WELD_COUNT : WORD ;
    RBT2_BT_CODE_NO : WORD ;
    RBT2_WELD_COUNT : WORD ;
    RBT3_BT_CODE_NO : WORD ;
    RBT3_WELD_COUNT : WORD ;
    RBT4_BT_CODE_NO : WORD ;
    RBT4_WELD_COUNT : WORD ;
    RBT5_BT_CODE_NO : WORD ;
    RBT5_WELD_COUNT : WORD ;
    RBT6_BT_CODE_NO : WORD ;
    RBT6_WELD_COUNT : WORD ;
    RBT7_BT_CODE_NO : WORD ;
    RBT7_WELD_COUNT : WORD ;
    RBT8_BT_CODE_NO : WORD ;
    RBT8_WELD_COUNT : WORD ;
    RBT9_BT_CODE_NO : WORD ;
    RBT9_WELD_COUNT : WORD ;
    RBT10_BT_CODE_NO : WORD ;
    RBT10_WELD_COUNT : WORD ;
    RBT11_BT_CODE_NO : WORD ;
    RBT11_WELD_COUNT : WORD ;
    RBT12_BT_CODE_NO : WORD ;
    RBT12_WELD_COUNT : WORD ;
    RBT13_BT_CODE_NO : WORD ;
    RBT13_WELD_COUNT : WORD ;
    RBT14_BT_CODE_NO : WORD ;
    RBT14_WELD_COUNT : WORD ;
    RBT15_BT_CODE_NO : WORD ;
    RBT15_WELD_COUNT : WORD ;
    RBT16_BT_CODE_NO : WORD ;
    RBT16_WELD_COUNT : WORD ;
    RBT17_BT_CODE_NO : WORD ;
    RBT17_WELD_COUNT : WORD ;
    RBT18_BT_CODE_NO : WORD ;
    RBT18_WELD_COUNT : WORD ;
    RBT19_BT_CODE_NO : WORD ;
    RBT19_WELD_COUNT : WORD ;
    RBT20_BT_CODE_NO : WORD ;
    RBT20_WELD_COUNT : WORD ;
    RBT21_BT_CODE_NO : WORD ;
    RBT21_WELD_COUNT : WORD ;
    RBT22_BT_CODE_NO : WORD ;
    RBT22_WELD_COUNT : WORD ;
    RBT23_BT_CODE_NO : WORD ;
    RBT23_WELD_COUNT : WORD ;
    RBT24_BT_CODE_NO : WORD ;
    RBT24_WELD_COUNT : WORD ;
    WELD_DETERMINES_RESULT : WORD ;
    WELD_CHECK_SUM : WORD ;
    SPARE1 : WORD ;
   END_STRUCT ;
   S711_WELD_BUFF_DATA1 : STRUCT
    STATION_MAIN : WORD ;
    DISTINCTION_LH_RH : WORD ;
    STAION_NUMBER : WORD ;
    VIN_NUMBER1 : WORD ;
    VIN_NUMBER2 : WORD ;
    VIN_NUMBER3 : WORD ;
    VIN_NUMBER4 : WORD ;
    SEQ_NUMBER1 : WORD ;
    SEQ_NUMBER2 : WORD ;
    RBT1_BT_CODE_NO : WORD ;
    RBT1_WELD_COUNT : WORD ;
    RBT2_BT_CODE_NO : WORD ;
    RBT2_WELD_COUNT : WORD ;
    RBT3_BT_CODE_NO : WORD ;
    RBT3_WELD_COUNT : WORD ;
    RBT4_BT_CODE_NO : WORD ;
    RBT4_WELD_COUNT : WORD ;
    RBT5_BT_CODE_NO : WORD ;
    RBT5_WELD_COUNT : WORD ;
    RBT6_BT_CODE_NO : WORD ;
    RBT6_WELD_COUNT : WORD ;
    RBT7_BT_CODE_NO : WORD ;
    RBT7_WELD_COUNT : WORD ;
    RBT8_BT_CODE_NO : WORD ;
    RBT8_WELD_COUNT : WORD ;
    RBT9_BT_CODE_NO : WORD ;
    RBT9_WELD_COUNT : WORD ;
    RBT10_BT_CODE_NO : WORD ;
    RBT10_WELD_COUNT : WORD ;
    RBT11_BT_CODE_NO : WORD ;
    RBT11_WELD_COUNT : WORD ;
    RBT12_BT_CODE_NO : WORD ;
    RBT12_WELD_COUNT : WORD ;
    RBT13_BT_CODE_NO : WORD ;
    RBT13_WELD_COUNT : WORD ;
    RBT14_BT_CODE_NO : WORD ;
    RBT14_WELD_COUNT : WORD ;
    RBT15_BT_CODE_NO : WORD ;
    RBT15_WELD_COUNT : WORD ;
    RBT16_BT_CODE_NO : WORD ;
    RBT16_WELD_COUNT : WORD ;
    RBT17_BT_CODE_NO : WORD ;
    RBT17_WELD_COUNT : WORD ;
    RBT18_BT_CODE_NO : WORD ;
    RBT18_WELD_COUNT : WORD ;
    RBT19_BT_CODE_NO : WORD ;
    RBT19_WELD_COUNT : WORD ;
    RBT20_BT_CODE_NO : WORD ;
    RBT20_WELD_COUNT : WORD ;
    RBT21_BT_CODE_NO : WORD ;
    RBT21_WELD_COUNT : WORD ;
    RBT22_BT_CODE_NO : WORD ;
    RBT22_WELD_COUNT : WORD ;
    RBT23_BT_CODE_NO : WORD ;
    RBT23_WELD_COUNT : WORD ;
    RBT24_BT_CODE_NO : WORD ;
    RBT24_WELD_COUNT : WORD ;
    WELD_DETERMINES_RESULT : WORD ;
    WELD_CHECK_SUM : WORD ;
    SPARE1 : WORD ;
   END_STRUCT ;
   S711_WELD_BUFF_DATA2 : STRUCT
    STATION_MAIN : WORD ;
    DISTINCTION_LH_RH : WORD ;
    STAION_NUMBER : WORD ;
    VIN_NUMBER1 : WORD ;
    VIN_NUMBER2 : WORD ;
    VIN_NUMBER3 : WORD ;
    VIN_NUMBER4 : WORD ;
    SEQ_NUMBER1 : WORD ;
    SEQ_NUMBER2 : WORD ;
    RBT1_BT_CODE_NO : WORD ;
    RBT1_WELD_COUNT : WORD ;
    RBT2_BT_CODE_NO : WORD ;
    RBT2_WELD_COUNT : WORD ;
    RBT3_BT_CODE_NO : WORD ;
    RBT3_WELD_COUNT : WORD ;
    RBT4_BT_CODE_NO : WORD ;
    RBT4_WELD_COUNT : WORD ;
    RBT5_BT_CODE_NO : WORD ;
    RBT5_WELD_COUNT : WORD ;
    RBT6_BT_CODE_NO : WORD ;
    RBT6_WELD_COUNT : WORD ;
    RBT7_BT_CODE_NO : WORD ;
    RBT7_WELD_COUNT : WORD ;
    RBT8_BT_CODE_NO : WORD ;
    RBT8_WELD_COUNT : WORD ;
    RBT9_BT_CODE_NO : WORD ;
    RBT9_WELD_COUNT : WORD ;
    RBT10_BT_CODE_NO : WORD ;
    RBT10_WELD_COUNT : WORD ;
    RBT11_BT_CODE_NO : WORD ;
    RBT11_WELD_COUNT : WORD ;
    RBT12_BT_CODE_NO : WORD ;
    RBT12_WELD_COUNT : WORD ;
    RBT13_BT_CODE_NO : WORD ;
    RBT13_WELD_COUNT : WORD ;
    RBT14_BT_CODE_NO : WORD ;
    RBT14_WELD_COUNT : WORD ;
    RBT15_BT_CODE_NO : WORD ;
    RBT15_WELD_COUNT : WORD ;
    RBT16_BT_CODE_NO : WORD ;
    RBT16_WELD_COUNT : WORD ;
    RBT17_BT_CODE_NO : WORD ;
    RBT17_WELD_COUNT : WORD ;
    RBT18_BT_CODE_NO : WORD ;
    RBT18_WELD_COUNT : WORD ;
    RBT19_BT_CODE_NO : WORD ;
    RBT19_WELD_COUNT : WORD ;
    RBT20_BT_CODE_NO : WORD ;
    RBT20_WELD_COUNT : WORD ;
    RBT21_BT_CODE_NO : WORD ;
    RBT21_WELD_COUNT : WORD ;
    RBT22_BT_CODE_NO : WORD ;
    RBT22_WELD_COUNT : WORD ;
    RBT23_BT_CODE_NO : WORD ;
    RBT23_WELD_COUNT : WORD ;
    RBT24_BT_CODE_NO : WORD ;
    RBT24_WELD_COUNT : WORD ;
    WELD_DETERMINES_RESULT : WORD ;
    WELD_CHECK_SUM : WORD ;
    SPARE1 : WORD ;
   END_STRUCT ;
   S711_WELD_BUFF_DATA3 : STRUCT
    STATION_MAIN : WORD ;
    DISTINCTION_LH_RH : WORD ;
    STAION_NUMBER : WORD ;
    VIN_NUMBER1 : WORD ;
    VIN_NUMBER2 : WORD ;
    VIN_NUMBER3 : WORD ;
    VIN_NUMBER4 : WORD ;
    SEQ_NUMBER1 : WORD ;
    SEQ_NUMBER2 : WORD ;
    RBT1_BT_CODE_NO : WORD ;
    RBT1_WELD_COUNT : WORD ;
    RBT2_BT_CODE_NO : WORD ;
    RBT2_WELD_COUNT : WORD ;
    RBT3_BT_CODE_NO : WORD ;
    RBT3_WELD_COUNT : WORD ;
    RBT4_BT_CODE_NO : WORD ;
    RBT4_WELD_COUNT : WORD ;
    RBT5_BT_CODE_NO : WORD ;
    RBT5_WELD_COUNT : WORD ;
    RBT6_BT_CODE_NO : WORD ;
    RBT6_WELD_COUNT : WORD ;
    RBT7_BT_CODE_NO : WORD ;
    RBT7_WELD_COUNT : WORD ;
    RBT8_BT_CODE_NO : WORD ;
    RBT8_WELD_COUNT : WORD ;
    RBT9_BT_CODE_NO : WORD ;
    RBT9_WELD_COUNT : WORD ;
    RBT10_BT_CODE_NO : WORD ;
    RBT10_WELD_COUNT : WORD ;
    RBT11_BT_CODE_NO : WORD ;
    RBT11_WELD_COUNT : WORD ;
    RBT12_BT_CODE_NO : WORD ;
    RBT12_WELD_COUNT : WORD ;
    RBT13_BT_CODE_NO : WORD ;
    RBT13_WELD_COUNT : WORD ;
    RBT14_BT_CODE_NO : WORD ;
    RBT14_WELD_COUNT : WORD ;
    RBT15_BT_CODE_NO : WORD ;
    RBT15_WELD_COUNT : WORD ;
    RBT16_BT_CODE_NO : WORD ;
    RBT16_WELD_COUNT : WORD ;
    RBT17_BT_CODE_NO : WORD ;
    RBT17_WELD_COUNT : WORD ;
    RBT18_BT_CODE_NO : WORD ;
    RBT18_WELD_COUNT : WORD ;
    RBT19_BT_CODE_NO : WORD ;
    RBT19_WELD_COUNT : WORD ;
    RBT20_BT_CODE_NO : WORD ;
    RBT20_WELD_COUNT : WORD ;
    RBT21_BT_CODE_NO : WORD ;
    RBT21_WELD_COUNT : WORD ;
    RBT22_BT_CODE_NO : WORD ;
    RBT22_WELD_COUNT : WORD ;
    RBT23_BT_CODE_NO : WORD ;
    RBT23_WELD_COUNT : WORD ;
    RBT24_BT_CODE_NO : WORD ;
    RBT24_WELD_COUNT : WORD ;
    WELD_DETERMINES_RESULT : WORD ;
    WELD_CHECK_SUM : WORD ;
    SPARE1 : WORD ;
   END_STRUCT ;
   S711_WELD_BUFF_DATA4 : STRUCT
    STATION_MAIN : WORD ;
    DISTINCTION_LH_RH : WORD ;
    STAION_NUMBER : WORD ;
    VIN_NUMBER1 : WORD ;
    VIN_NUMBER2 : WORD ;
    VIN_NUMBER3 : WORD ;
    VIN_NUMBER4 : WORD ;
    SEQ_NUMBER1 : WORD ;
    SEQ_NUMBER2 : WORD ;
    RBT1_BT_CODE_NO : WORD ;
    RBT1_WELD_COUNT : WORD ;
    RBT2_BT_CODE_NO : WORD ;
    RBT2_WELD_COUNT : WORD ;
    RBT3_BT_CODE_NO : WORD ;
    RBT3_WELD_COUNT : WORD ;
    RBT4_BT_CODE_NO : WORD ;
    RBT4_WELD_COUNT : WORD ;
    RBT5_BT_CODE_NO : WORD ;
    RBT5_WELD_COUNT : WORD ;
    RBT6_BT_CODE_NO : WORD ;
    RBT6_WELD_COUNT : WORD ;
    RBT7_BT_CODE_NO : WORD ;
    RBT7_WELD_COUNT : WORD ;
    RBT8_BT_CODE_NO : WORD ;
    RBT8_WELD_COUNT : WORD ;
    RBT9_BT_CODE_NO : WORD ;
    RBT9_WELD_COUNT : WORD ;
    RBT10_BT_CODE_NO : WORD ;
    RBT10_WELD_COUNT : WORD ;
    RBT11_BT_CODE_NO : WORD ;
    RBT11_WELD_COUNT : WORD ;
    RBT12_BT_CODE_NO : WORD ;
    RBT12_WELD_COUNT : WORD ;
    RBT13_BT_CODE_NO : WORD ;
    RBT13_WELD_COUNT : WORD ;
    RBT14_BT_CODE_NO : WORD ;
    RBT14_WELD_COUNT : WORD ;
    RBT15_BT_CODE_NO : WORD ;
    RBT15_WELD_COUNT : WORD ;
    RBT16_BT_CODE_NO : WORD ;
    RBT16_WELD_COUNT : WORD ;
    RBT17_BT_CODE_NO : WORD ;
    RBT17_WELD_COUNT : WORD ;
    RBT18_BT_CODE_NO : WORD ;
    RBT18_WELD_COUNT : WORD ;
    RBT19_BT_CODE_NO : WORD ;
    RBT19_WELD_COUNT : WORD ;
    RBT20_BT_CODE_NO : WORD ;
    RBT20_WELD_COUNT : WORD ;
    RBT21_BT_CODE_NO : WORD ;
    RBT21_WELD_COUNT : WORD ;
    RBT22_BT_CODE_NO : WORD ;
    RBT22_WELD_COUNT : WORD ;
    RBT23_BT_CODE_NO : WORD ;
    RBT23_WELD_COUNT : WORD ;
    RBT24_BT_CODE_NO : WORD ;
    RBT24_WELD_COUNT : WORD ;
    WELD_DETERMINES_RESULT : WORD ;
    WELD_CHECK_SUM : WORD ;
    SPARE1 : WORD ;
   END_STRUCT ;
   S711_WELD_BUFF_DATA5 : STRUCT
    STATION_MAIN : WORD ;
    DISTINCTION_LH_RH : WORD ;
    STAION_NUMBER : WORD ;
    VIN_NUMBER1 : WORD ;
    VIN_NUMBER2 : WORD ;
    VIN_NUMBER3 : WORD ;
    VIN_NUMBER4 : WORD ;
    SEQ_NUMBER1 : WORD ;
    SEQ_NUMBER2 : WORD ;
    RBT1_BT_CODE_NO : WORD ;
    RBT1_WELD_COUNT : WORD ;
    RBT2_BT_CODE_NO : WORD ;
    RBT2_WELD_COUNT : WORD ;
    RBT3_BT_CODE_NO : WORD ;
    RBT3_WELD_COUNT : WORD ;
    RBT4_BT_CODE_NO : WORD ;
    RBT4_WELD_COUNT : WORD ;
    RBT5_BT_CODE_NO : WORD ;
    RBT5_WELD_COUNT : WORD ;
    RBT6_BT_CODE_NO : WORD ;
    RBT6_WELD_COUNT : WORD ;
    RBT7_BT_CODE_NO : WORD ;
    RBT7_WELD_COUNT : WORD ;
    RBT8_BT_CODE_NO : WORD ;
    RBT8_WELD_COUNT : WORD ;
    RBT9_BT_CODE_NO : WORD ;
    RBT9_WELD_COUNT : WORD ;
    RBT10_BT_CODE_NO : WORD ;
    RBT10_WELD_COUNT : WORD ;
    RBT11_BT_CODE_NO : WORD ;
    RBT11_WELD_COUNT : WORD ;
    RBT12_BT_CODE_NO : WORD ;
    RBT12_WELD_COUNT : WORD ;
    RBT13_BT_CODE_NO : WORD ;
    RBT13_WELD_COUNT : WORD ;
    RBT14_BT_CODE_NO : WORD ;
    RBT14_WELD_COUNT : WORD ;
    RBT15_BT_CODE_NO : WORD ;
    RBT15_WELD_COUNT : WORD ;
    RBT16_BT_CODE_NO : WORD ;
    RBT16_WELD_COUNT : WORD ;
    RBT17_BT_CODE_NO : WORD ;
    RBT17_WELD_COUNT : WORD ;
    RBT18_BT_CODE_NO : WORD ;
    RBT18_WELD_COUNT : WORD ;
    RBT19_BT_CODE_NO : WORD ;
    RBT19_WELD_COUNT : WORD ;
    RBT20_BT_CODE_NO : WORD ;
    RBT20_WELD_COUNT : WORD ;
    RBT21_BT_CODE_NO : WORD ;
    RBT21_WELD_COUNT : WORD ;
    RBT22_BT_CODE_NO : WORD ;
    RBT22_WELD_COUNT : WORD ;
    RBT23_BT_CODE_NO : WORD ;
    RBT23_WELD_COUNT : WORD ;
    RBT24_BT_CODE_NO : WORD ;
    RBT24_WELD_COUNT : WORD ;
    WELD_DETERMINES_RESULT : WORD ;
    WELD_CHECK_SUM : WORD ;
    SPARE1 : WORD ;
   END_STRUCT ;
   S711_WELD_BUFF_DATA6 : STRUCT
    STATION_MAIN : WORD ;
    DISTINCTION_LH_RH : WORD ;
    STAION_NUMBER : WORD ;
    VIN_NUMBER1 : WORD ;
    VIN_NUMBER2 : WORD ;
    VIN_NUMBER3 : WORD ;
    VIN_NUMBER4 : WORD ;
    SEQ_NUMBER1 : WORD ;
    SEQ_NUMBER2 : WORD ;
    RBT1_BT_CODE_NO : WORD ;
    RBT1_WELD_COUNT : WORD ;
    RBT2_BT_CODE_NO : WORD ;
    RBT2_WELD_COUNT : WORD ;
    RBT3_BT_CODE_NO : WORD ;
    RBT3_WELD_COUNT : WORD ;
    RBT4_BT_CODE_NO : WORD ;
    RBT4_WELD_COUNT : WORD ;
    RBT5_BT_CODE_NO : WORD ;
    RBT5_WELD_COUNT : WORD ;
    RBT6_BT_CODE_NO : WORD ;
    RBT6_WELD_COUNT : WORD ;
    RBT7_BT_CODE_NO : WORD ;
    RBT7_WELD_COUNT : WORD ;
    RBT8_BT_CODE_NO : WORD ;
    RBT8_WELD_COUNT : WORD ;
    RBT9_BT_CODE_NO : WORD ;
    RBT9_WELD_COUNT : WORD ;
    RBT10_BT_CODE_NO : WORD ;
    RBT10_WELD_COUNT : WORD ;
    RBT11_BT_CODE_NO : WORD ;
    RBT11_WELD_COUNT : WORD ;
    RBT12_BT_CODE_NO : WORD ;
    RBT12_WELD_COUNT : WORD ;
    RBT13_BT_CODE_NO : WORD ;
    RBT13_WELD_COUNT : WORD ;
    RBT14_BT_CODE_NO : WORD ;
    RBT14_WELD_COUNT : WORD ;
    RBT15_BT_CODE_NO : WORD ;
    RBT15_WELD_COUNT : WORD ;
    RBT16_BT_CODE_NO : WORD ;
    RBT16_WELD_COUNT : WORD ;
    RBT17_BT_CODE_NO : WORD ;
    RBT17_WELD_COUNT : WORD ;
    RBT18_BT_CODE_NO : WORD ;
    RBT18_WELD_COUNT : WORD ;
    RBT19_BT_CODE_NO : WORD ;
    RBT19_WELD_COUNT : WORD ;
    RBT20_BT_CODE_NO : WORD ;
    RBT20_WELD_COUNT : WORD ;
    RBT21_BT_CODE_NO : WORD ;
    RBT21_WELD_COUNT : WORD ;
    RBT22_BT_CODE_NO : WORD ;
    RBT22_WELD_COUNT : WORD ;
    RBT23_BT_CODE_NO : WORD ;
    RBT23_WELD_COUNT : WORD ;
    RBT24_BT_CODE_NO : WORD ;
    RBT24_WELD_COUNT : WORD ;
    WELD_DETERMINES_RESULT : WORD ;
    WELD_CHECK_SUM : WORD ;
    SPARE1 : WORD ;
   END_STRUCT ;
   S711_WELD_BUFF_DATA7 : STRUCT
    STATION_MAIN : WORD ;
    DISTINCTION_LH_RH : WORD ;
    STAION_NUMBER : WORD ;
    VIN_NUMBER1 : WORD ;
    VIN_NUMBER2 : WORD ;
    VIN_NUMBER3 : WORD ;
    VIN_NUMBER4 : WORD ;
    SEQ_NUMBER1 : WORD ;
    SEQ_NUMBER2 : WORD ;
    RBT1_BT_CODE_NO : WORD ;
    RBT1_WELD_COUNT : WORD ;
    RBT2_BT_CODE_NO : WORD ;
    RBT2_WELD_COUNT : WORD ;
    RBT3_BT_CODE_NO : WORD ;
    RBT3_WELD_COUNT : WORD ;
    RBT4_BT_CODE_NO : WORD ;
    RBT4_WELD_COUNT : WORD ;
    RBT5_BT_CODE_NO : WORD ;
    RBT5_WELD_COUNT : WORD ;
    RBT6_BT_CODE_NO : WORD ;
    RBT6_WELD_COUNT : WORD ;
    RBT7_BT_CODE_NO : WORD ;
    RBT7_WELD_COUNT : WORD ;
    RBT8_BT_CODE_NO : WORD ;
    RBT8_WELD_COUNT : WORD ;
    RBT9_BT_CODE_NO : WORD ;
    RBT9_WELD_COUNT : WORD ;
    RBT10_BT_CODE_NO : WORD ;
    RBT10_WELD_COUNT : WORD ;
    RBT11_BT_CODE_NO : WORD ;
    RBT11_WELD_COUNT : WORD ;
    RBT12_BT_CODE_NO : WORD ;
    RBT12_WELD_COUNT : WORD ;
    RBT13_BT_CODE_NO : WORD ;
    RBT13_WELD_COUNT : WORD ;
    RBT14_BT_CODE_NO : WORD ;
    RBT14_WELD_COUNT : WORD ;
    RBT15_BT_CODE_NO : WORD ;
    RBT15_WELD_COUNT : WORD ;
    RBT16_BT_CODE_NO : WORD ;
    RBT16_WELD_COUNT : WORD ;
    RBT17_BT_CODE_NO : WORD ;
    RBT17_WELD_COUNT : WORD ;
    RBT18_BT_CODE_NO : WORD ;
    RBT18_WELD_COUNT : WORD ;
    RBT19_BT_CODE_NO : WORD ;
    RBT19_WELD_COUNT : WORD ;
    RBT20_BT_CODE_NO : WORD ;
    RBT20_WELD_COUNT : WORD ;
    RBT21_BT_CODE_NO : WORD ;
    RBT21_WELD_COUNT : WORD ;
    RBT22_BT_CODE_NO : WORD ;
    RBT22_WELD_COUNT : WORD ;
    RBT23_BT_CODE_NO : WORD ;
    RBT23_WELD_COUNT : WORD ;
    RBT24_BT_CODE_NO : WORD ;
    RBT24_WELD_COUNT : WORD ;
    WELD_DETERMINES_RESULT : WORD ;
    WELD_CHECK_SUM : WORD ;
    SPARE1 : WORD ;
   END_STRUCT ;
   S711_WELD_BUFF_DATA8 : STRUCT
    STATION_MAIN : WORD ;
    DISTINCTION_LH_RH : WORD ;
    STAION_NUMBER : WORD ;
    VIN_NUMBER1 : WORD ;
    VIN_NUMBER2 : WORD ;
    VIN_NUMBER3 : WORD ;
    VIN_NUMBER4 : WORD ;
    SEQ_NUMBER1 : WORD ;
    SEQ_NUMBER2 : WORD ;
    RBT1_BT_CODE_NO : WORD ;
    RBT1_WELD_COUNT : WORD ;
    RBT2_BT_CODE_NO : WORD ;
    RBT2_WELD_COUNT : WORD ;
    RBT3_BT_CODE_NO : WORD ;
    RBT3_WELD_COUNT : WORD ;
    RBT4_BT_CODE_NO : WORD ;
    RBT4_WELD_COUNT : WORD ;
    RBT5_BT_CODE_NO : WORD ;
    RBT5_WELD_COUNT : WORD ;
    RBT6_BT_CODE_NO : WORD ;
    RBT6_WELD_COUNT : WORD ;
    RBT7_BT_CODE_NO : WORD ;
    RBT7_WELD_COUNT : WORD ;
    RBT8_BT_CODE_NO : WORD ;
    RBT8_WELD_COUNT : WORD ;
    RBT9_BT_CODE_NO : WORD ;
    RBT9_WELD_COUNT : WORD ;
    RBT10_BT_CODE_NO : WORD ;
    RBT10_WELD_COUNT : WORD ;
    RBT11_BT_CODE_NO : WORD ;
    RBT11_WELD_COUNT : WORD ;
    RBT12_BT_CODE_NO : WORD ;
    RBT12_WELD_COUNT : WORD ;
    RBT13_BT_CODE_NO : WORD ;
    RBT13_WELD_COUNT : WORD ;
    RBT14_BT_CODE_NO : WORD ;
    RBT14_WELD_COUNT : WORD ;
    RBT15_BT_CODE_NO : WORD ;
    RBT15_WELD_COUNT : WORD ;
    RBT16_BT_CODE_NO : WORD ;
    RBT16_WELD_COUNT : WORD ;
    RBT17_BT_CODE_NO : WORD ;
    RBT17_WELD_COUNT : WORD ;
    RBT18_BT_CODE_NO : WORD ;
    RBT18_WELD_COUNT : WORD ;
    RBT19_BT_CODE_NO : WORD ;
    RBT19_WELD_COUNT : WORD ;
    RBT20_BT_CODE_NO : WORD ;
    RBT20_WELD_COUNT : WORD ;
    RBT21_BT_CODE_NO : WORD ;
    RBT21_WELD_COUNT : WORD ;
    RBT22_BT_CODE_NO : WORD ;
    RBT22_WELD_COUNT : WORD ;
    RBT23_BT_CODE_NO : WORD ;
    RBT23_WELD_COUNT : WORD ;
    RBT24_BT_CODE_NO : WORD ;
    RBT24_WELD_COUNT : WORD ;
    WELD_DETERMINES_RESULT : WORD ;
    WELD_CHECK_SUM : WORD ;
    SPARE1 : WORD ;
   END_STRUCT ;
   S711_WELD_BUFF_DATA9 : STRUCT
    STATION_MAIN : WORD ;
    DISTINCTION_LH_RH : WORD ;
    STAION_NUMBER : WORD ;
    VIN_NUMBER1 : WORD ;
    VIN_NUMBER2 : WORD ;
    VIN_NUMBER3 : WORD ;
    VIN_NUMBER4 : WORD ;
    SEQ_NUMBER1 : WORD ;
    SEQ_NUMBER2 : WORD ;
    RBT1_BT_CODE_NO : WORD ;
    RBT1_WELD_COUNT : WORD ;
    RBT2_BT_CODE_NO : WORD ;
    RBT2_WELD_COUNT : WORD ;
    RBT3_BT_CODE_NO : WORD ;
    RBT3_WELD_COUNT : WORD ;
    RBT4_BT_CODE_NO : WORD ;
    RBT4_WELD_COUNT : WORD ;
    RBT5_BT_CODE_NO : WORD ;
    RBT5_WELD_COUNT : WORD ;
    RBT6_BT_CODE_NO : WORD ;
    RBT6_WELD_COUNT : WORD ;
    RBT7_BT_CODE_NO : WORD ;
    RBT7_WELD_COUNT : WORD ;
    RBT8_BT_CODE_NO : WORD ;
    RBT8_WELD_COUNT : WORD ;
    RBT9_BT_CODE_NO : WORD ;
    RBT9_WELD_COUNT : WORD ;
    RBT10_BT_CODE_NO : WORD ;
    RBT10_WELD_COUNT : WORD ;
    RBT11_BT_CODE_NO : WORD ;
    RBT11_WELD_COUNT : WORD ;
    RBT12_BT_CODE_NO : WORD ;
    RBT12_WELD_COUNT : WORD ;
    RBT13_BT_CODE_NO : WORD ;
    RBT13_WELD_COUNT : WORD ;
    RBT14_BT_CODE_NO : WORD ;
    RBT14_WELD_COUNT : WORD ;
    RBT15_BT_CODE_NO : WORD ;
    RBT15_WELD_COUNT : WORD ;
    RBT16_BT_CODE_NO : WORD ;
    RBT16_WELD_COUNT : WORD ;
    RBT17_BT_CODE_NO : WORD ;
    RBT17_WELD_COUNT : WORD ;
    RBT18_BT_CODE_NO : WORD ;
    RBT18_WELD_COUNT : WORD ;
    RBT19_BT_CODE_NO : WORD ;
    RBT19_WELD_COUNT : WORD ;
    RBT20_BT_CODE_NO : WORD ;
    RBT20_WELD_COUNT : WORD ;
    RBT21_BT_CODE_NO : WORD ;
    RBT21_WELD_COUNT : WORD ;
    RBT22_BT_CODE_NO : WORD ;
    RBT22_WELD_COUNT : WORD ;
    RBT23_BT_CODE_NO : WORD ;
    RBT23_WELD_COUNT : WORD ;
    RBT24_BT_CODE_NO : WORD ;
    RBT24_WELD_COUNT : WORD ;
    WELD_DETERMINES_RESULT : WORD ;
    WELD_CHECK_SUM : WORD ;
    SPARE1 : WORD ;
   END_STRUCT ;
   S711_WELD_BUFF_DATA10 : STRUCT
    STATION_MAIN : WORD ;
    DISTINCTION_LH_RH : WORD ;
    STAION_NUMBER : WORD ;
    VIN_NUMBER1 : WORD ;
    VIN_NUMBER2 : WORD ;
    VIN_NUMBER3 : WORD ;
    VIN_NUMBER4 : WORD ;
    SEQ_NUMBER1 : WORD ;
    SEQ_NUMBER2 : WORD ;
    RBT1_BT_CODE_NO : WORD ;
    RBT1_WELD_COUNT : WORD ;
    RBT2_BT_CODE_NO : WORD ;
    RBT2_WELD_COUNT : WORD ;
    RBT3_BT_CODE_NO : WORD ;
    RBT3_WELD_COUNT : WORD ;
    RBT4_BT_CODE_NO : WORD ;
    RBT4_WELD_COUNT : WORD ;
    RBT5_BT_CODE_NO : WORD ;
    RBT5_WELD_COUNT : WORD ;
    RBT6_BT_CODE_NO : WORD ;
    RBT6_WELD_COUNT : WORD ;
    RBT7_BT_CODE_NO : WORD ;
    RBT7_WELD_COUNT : WORD ;
    RBT8_BT_CODE_NO : WORD ;
    RBT8_WELD_COUNT : WORD ;
    RBT9_BT_CODE_NO : WORD ;
    RBT9_WELD_COUNT : WORD ;
    RBT10_BT_CODE_NO : WORD ;
    RBT10_WELD_COUNT : WORD ;
    RBT11_BT_CODE_NO : WORD ;
    RBT11_WELD_COUNT : WORD ;
    RBT12_BT_CODE_NO : WORD ;
    RBT12_WELD_COUNT : WORD ;
    RBT13_BT_CODE_NO : WORD ;
    RBT13_WELD_COUNT : WORD ;
    RBT14_BT_CODE_NO : WORD ;
    RBT14_WELD_COUNT : WORD ;
    RBT15_BT_CODE_NO : WORD ;
    RBT15_WELD_COUNT : WORD ;
    RBT16_BT_CODE_NO : WORD ;
    RBT16_WELD_COUNT : WORD ;
    RBT17_BT_CODE_NO : WORD ;
    RBT17_WELD_COUNT : WORD ;
    RBT18_BT_CODE_NO : WORD ;
    RBT18_WELD_COUNT : WORD ;
    RBT19_BT_CODE_NO : WORD ;
    RBT19_WELD_COUNT : WORD ;
    RBT20_BT_CODE_NO : WORD ;
    RBT20_WELD_COUNT : WORD ;
    RBT21_BT_CODE_NO : WORD ;
    RBT21_WELD_COUNT : WORD ;
    RBT22_BT_CODE_NO : WORD ;
    RBT22_WELD_COUNT : WORD ;
    RBT23_BT_CODE_NO : WORD ;
    RBT23_WELD_COUNT : WORD ;
    RBT24_BT_CODE_NO : WORD ;
    RBT24_WELD_COUNT : WORD ;
    WELD_DETERMINES_RESULT : WORD ;
    WELD_CHECK_SUM : WORD ;
    SPARE1 : WORD ;
   END_STRUCT ;
   S711_WELD_BUFF_DATA11 : STRUCT
    STATION_MAIN : WORD ;
    DISTINCTION_LH_RH : WORD ;
    STAION_NUMBER : WORD ;
    VIN_NUMBER1 : WORD ;
    VIN_NUMBER2 : WORD ;
    VIN_NUMBER3 : WORD ;
    VIN_NUMBER4 : WORD ;
    SEQ_NUMBER1 : WORD ;
    SEQ_NUMBER2 : WORD ;
    RBT1_BT_CODE_NO : WORD ;
    RBT1_WELD_COUNT : WORD ;
    RBT2_BT_CODE_NO : WORD ;
    RBT2_WELD_COUNT : WORD ;
    RBT3_BT_CODE_NO : WORD ;
    RBT3_WELD_COUNT : WORD ;
    RBT4_BT_CODE_NO : WORD ;
    RBT4_WELD_COUNT : WORD ;
    RBT5_BT_CODE_NO : WORD ;
    RBT5_WELD_COUNT : WORD ;
    RBT6_BT_CODE_NO : WORD ;
    RBT6_WELD_COUNT : WORD ;
    RBT7_BT_CODE_NO : WORD ;
    RBT7_WELD_COUNT : WORD ;
    RBT8_BT_CODE_NO : WORD ;
    RBT8_WELD_COUNT : WORD ;
    RBT9_BT_CODE_NO : WORD ;
    RBT9_WELD_COUNT : WORD ;
    RBT10_BT_CODE_NO : WORD ;
    RBT10_WELD_COUNT : WORD ;
    RBT11_BT_CODE_NO : WORD ;
    RBT11_WELD_COUNT : WORD ;
    RBT12_BT_CODE_NO : WORD ;
    RBT12_WELD_COUNT : WORD ;
    RBT13_BT_CODE_NO : WORD ;
    RBT13_WELD_COUNT : WORD ;
    RBT14_BT_CODE_NO : WORD ;
    RBT14_WELD_COUNT : WORD ;
    RBT15_BT_CODE_NO : WORD ;
    RBT15_WELD_COUNT : WORD ;
    RBT16_BT_CODE_NO : WORD ;
    RBT16_WELD_COUNT : WORD ;
    RBT17_BT_CODE_NO : WORD ;
    RBT17_WELD_COUNT : WORD ;
    RBT18_BT_CODE_NO : WORD ;
    RBT18_WELD_COUNT : WORD ;
    RBT19_BT_CODE_NO : WORD ;
    RBT19_WELD_COUNT : WORD ;
    RBT20_BT_CODE_NO : WORD ;
    RBT20_WELD_COUNT : WORD ;
    RBT21_BT_CODE_NO : WORD ;
    RBT21_WELD_COUNT : WORD ;
    RBT22_BT_CODE_NO : WORD ;
    RBT22_WELD_COUNT : WORD ;
    RBT23_BT_CODE_NO : WORD ;
    RBT23_WELD_COUNT : WORD ;
    RBT24_BT_CODE_NO : WORD ;
    RBT24_WELD_COUNT : WORD ;
    WELD_DETERMINES_RESULT : WORD ;
    WELD_CHECK_SUM : WORD ;
    SPARE1 : WORD ;
   END_STRUCT ;
   S711_WELD_BUFF_DATA21 : STRUCT
    STATION_MAIN : WORD ;
    DISTINCTION_LH_RH : WORD ;
    STAION_NUMBER : WORD ;
    VIN_NUMBER1 : WORD ;
    VIN_NUMBER2 : WORD ;
    VIN_NUMBER3 : WORD ;
    VIN_NUMBER4 : WORD ;
    SEQ_NUMBER1 : WORD ;
    SEQ_NUMBER2 : WORD ;
    RBT1_BT_CODE_NO : WORD ;
    RBT1_WELD_COUNT : WORD ;
    RBT2_BT_CODE_NO : WORD ;
    RBT2_WELD_COUNT : WORD ;
    RBT3_BT_CODE_NO : WORD ;
    RBT3_WELD_COUNT : WORD ;
    RBT4_BT_CODE_NO : WORD ;
    RBT4_WELD_COUNT : WORD ;
    RBT5_BT_CODE_NO : WORD ;
    RBT5_WELD_COUNT : WORD ;
    RBT6_BT_CODE_NO : WORD ;
    RBT6_WELD_COUNT : WORD ;
    RBT7_BT_CODE_NO : WORD ;
    RBT7_WELD_COUNT : WORD ;
    RBT8_BT_CODE_NO : WORD ;
    RBT8_WELD_COUNT : WORD ;
    RBT9_BT_CODE_NO : WORD ;
    RBT9_WELD_COUNT : WORD ;
    RBT10_BT_CODE_NO : WORD ;
    RBT10_WELD_COUNT : WORD ;
    RBT11_BT_CODE_NO : WORD ;
    RBT11_WELD_COUNT : WORD ;
    RBT12_BT_CODE_NO : WORD ;
    RBT12_WELD_COUNT : WORD ;
    RBT13_BT_CODE_NO : WORD ;
    RBT13_WELD_COUNT : WORD ;
    RBT14_BT_CODE_NO : WORD ;
    RBT14_WELD_COUNT : WORD ;
    RBT15_BT_CODE_NO : WORD ;
    RBT15_WELD_COUNT : WORD ;
    RBT16_BT_CODE_NO : WORD ;
    RBT16_WELD_COUNT : WORD ;
    RBT17_BT_CODE_NO : WORD ;
    RBT17_WELD_COUNT : WORD ;
    RBT18_BT_CODE_NO : WORD ;
    RBT18_WELD_COUNT : WORD ;
    RBT19_BT_CODE_NO : WORD ;
    RBT19_WELD_COUNT : WORD ;
    RBT20_BT_CODE_NO : WORD ;
    RBT20_WELD_COUNT : WORD ;
    RBT21_BT_CODE_NO : WORD ;
    RBT21_WELD_COUNT : WORD ;
    RBT22_BT_CODE_NO : WORD ;
    RBT22_WELD_COUNT : WORD ;
    RBT23_BT_CODE_NO : WORD ;
    RBT23_WELD_COUNT : WORD ;
    RBT24_BT_CODE_NO : WORD ;
    RBT24_WELD_COUNT : WORD ;
    WELD_DETERMINES_RESULT : WORD ;
    WELD_CHECK_SUM : WORD ;
    SPARE1 : WORD ;
   END_STRUCT ;
   S711_WELD_BUFF_DATA31 : STRUCT
    STATION_MAIN : WORD ;
    DISTINCTION_LH_RH : WORD ;
    STAION_NUMBER : WORD ;
    VIN_NUMBER1 : WORD ;
    VIN_NUMBER2 : WORD ;
    VIN_NUMBER3 : WORD ;
    VIN_NUMBER4 : WORD ;
    SEQ_NUMBER1 : WORD ;
    SEQ_NUMBER2 : WORD ;
    RBT1_BT_CODE_NO : WORD ;
    RBT1_WELD_COUNT : WORD ;
    RBT2_BT_CODE_NO : WORD ;
    RBT2_WELD_COUNT : WORD ;
    RBT3_BT_CODE_NO : WORD ;
    RBT3_WELD_COUNT : WORD ;
    RBT4_BT_CODE_NO : WORD ;
    RBT4_WELD_COUNT : WORD ;
    RBT5_BT_CODE_NO : WORD ;
    RBT5_WELD_COUNT : WORD ;
    RBT6_BT_CODE_NO : WORD ;
    RBT6_WELD_COUNT : WORD ;
    RBT7_BT_CODE_NO : WORD ;
    RBT7_WELD_COUNT : WORD ;
    RBT8_BT_CODE_NO : WORD ;
    RBT8_WELD_COUNT : WORD ;
    RBT9_BT_CODE_NO : WORD ;
    RBT9_WELD_COUNT : WORD ;
    RBT10_BT_CODE_NO : WORD ;
    RBT10_WELD_COUNT : WORD ;
    RBT11_BT_CODE_NO : WORD ;
    RBT11_WELD_COUNT : WORD ;
    RBT12_BT_CODE_NO : WORD ;
    RBT12_WELD_COUNT : WORD ;
    RBT13_BT_CODE_NO : WORD ;
    RBT13_WELD_COUNT : WORD ;
    RBT14_BT_CODE_NO : WORD ;
    RBT14_WELD_COUNT : WORD ;
    RBT15_BT_CODE_NO : WORD ;
    RBT15_WELD_COUNT : WORD ;
    RBT16_BT_CODE_NO : WORD ;
    RBT16_WELD_COUNT : WORD ;
    RBT17_BT_CODE_NO : WORD ;
    RBT17_WELD_COUNT : WORD ;
    RBT18_BT_CODE_NO : WORD ;
    RBT18_WELD_COUNT : WORD ;
    RBT19_BT_CODE_NO : WORD ;
    RBT19_WELD_COUNT : WORD ;
    RBT20_BT_CODE_NO : WORD ;
    RBT20_WELD_COUNT : WORD ;
    RBT21_BT_CODE_NO : WORD ;
    RBT21_WELD_COUNT : WORD ;
    RBT22_BT_CODE_NO : WORD ;
    RBT22_WELD_COUNT : WORD ;
    RBT23_BT_CODE_NO : WORD ;
    RBT23_WELD_COUNT : WORD ;
    RBT24_BT_CODE_NO : WORD ;
    RBT24_WELD_COUNT : WORD ;
    WELD_DETERMINES_RESULT : WORD ;
    WELD_CHECK_SUM : WORD ;
    SPARE1 : WORD ;
   END_STRUCT ;
   S711_WELD_BUFF_DATA41 : STRUCT
    STATION_MAIN : WORD ;
    DISTINCTION_LH_RH : WORD ;
    STAION_NUMBER : WORD ;
    VIN_NUMBER1 : WORD ;
    VIN_NUMBER2 : WORD ;
    VIN_NUMBER3 : WORD ;
    VIN_NUMBER4 : WORD ;
    SEQ_NUMBER1 : WORD ;
    SEQ_NUMBER2 : WORD ;
    RBT1_BT_CODE_NO : WORD ;
    RBT1_WELD_COUNT : WORD ;
    RBT2_BT_CODE_NO : WORD ;
    RBT2_WELD_COUNT : WORD ;
    RBT3_BT_CODE_NO : WORD ;
    RBT3_WELD_COUNT : WORD ;
    RBT4_BT_CODE_NO : WORD ;
    RBT4_WELD_COUNT : WORD ;
    RBT5_BT_CODE_NO : WORD ;
    RBT5_WELD_COUNT : WORD ;
    RBT6_BT_CODE_NO : WORD ;
    RBT6_WELD_COUNT : WORD ;
    RBT7_BT_CODE_NO : WORD ;
    RBT7_WELD_COUNT : WORD ;
    RBT8_BT_CODE_NO : WORD ;
    RBT8_WELD_COUNT : WORD ;
    RBT9_BT_CODE_NO : WORD ;
    RBT9_WELD_COUNT : WORD ;
    RBT10_BT_CODE_NO : WORD ;
    RBT10_WELD_COUNT : WORD ;
    RBT11_BT_CODE_NO : WORD ;
    RBT11_WELD_COUNT : WORD ;
    RBT12_BT_CODE_NO : WORD ;
    RBT12_WELD_COUNT : WORD ;
    RBT13_BT_CODE_NO : WORD ;
    RBT13_WELD_COUNT : WORD ;
    RBT14_BT_CODE_NO : WORD ;
    RBT14_WELD_COUNT : WORD ;
    RBT15_BT_CODE_NO : WORD ;
    RBT15_WELD_COUNT : WORD ;
    RBT16_BT_CODE_NO : WORD ;
    RBT16_WELD_COUNT : WORD ;
    RBT17_BT_CODE_NO : WORD ;
    RBT17_WELD_COUNT : WORD ;
    RBT18_BT_CODE_NO : WORD ;
    RBT18_WELD_COUNT : WORD ;
    RBT19_BT_CODE_NO : WORD ;
    RBT19_WELD_COUNT : WORD ;
    RBT20_BT_CODE_NO : WORD ;
    RBT20_WELD_COUNT : WORD ;
    RBT21_BT_CODE_NO : WORD ;
    RBT21_WELD_COUNT : WORD ;
    RBT22_BT_CODE_NO : WORD ;
    RBT22_WELD_COUNT : WORD ;
    RBT23_BT_CODE_NO : WORD ;
    RBT23_WELD_COUNT : WORD ;
    RBT24_BT_CODE_NO : WORD ;
    RBT24_WELD_COUNT : WORD ;
    WELD_DETERMINES_RESULT : WORD ;
    WELD_CHECK_SUM : WORD ;
    SPARE1 : WORD ;
   END_STRUCT ;
   S711_WELD_BUFF_DATA51 : STRUCT
    STATION_MAIN : WORD ;
    DISTINCTION_LH_RH : WORD ;
    STAION_NUMBER : WORD ;
    VIN_NUMBER1 : WORD ;
    VIN_NUMBER2 : WORD ;
    VIN_NUMBER3 : WORD ;
    VIN_NUMBER4 : WORD ;
    SEQ_NUMBER1 : WORD ;
    SEQ_NUMBER2 : WORD ;
    RBT1_BT_CODE_NO : WORD ;
    RBT1_WELD_COUNT : WORD ;
    RBT2_BT_CODE_NO : WORD ;
    RBT2_WELD_COUNT : WORD ;
    RBT3_BT_CODE_NO : WORD ;
    RBT3_WELD_COUNT : WORD ;
    RBT4_BT_CODE_NO : WORD ;
    RBT4_WELD_COUNT : WORD ;
    RBT5_BT_CODE_NO : WORD ;
    RBT5_WELD_COUNT : WORD ;
    RBT6_BT_CODE_NO : WORD ;
    RBT6_WELD_COUNT : WORD ;
    RBT7_BT_CODE_NO : WORD ;
    RBT7_WELD_COUNT : WORD ;
    RBT8_BT_CODE_NO : WORD ;
    RBT8_WELD_COUNT : WORD ;
    RBT9_BT_CODE_NO : WORD ;
    RBT9_WELD_COUNT : WORD ;
    RBT10_BT_CODE_NO : WORD ;
    RBT10_WELD_COUNT : WORD ;
    RBT11_BT_CODE_NO : WORD ;
    RBT11_WELD_COUNT : WORD ;
    RBT12_BT_CODE_NO : WORD ;
    RBT12_WELD_COUNT : WORD ;
    RBT13_BT_CODE_NO : WORD ;
    RBT13_WELD_COUNT : WORD ;
    RBT14_BT_CODE_NO : WORD ;
    RBT14_WELD_COUNT : WORD ;
    RBT15_BT_CODE_NO : WORD ;
    RBT15_WELD_COUNT : WORD ;
    RBT16_BT_CODE_NO : WORD ;
    RBT16_WELD_COUNT : WORD ;
    RBT17_BT_CODE_NO : WORD ;
    RBT17_WELD_COUNT : WORD ;
    RBT18_BT_CODE_NO : WORD ;
    RBT18_WELD_COUNT : WORD ;
    RBT19_BT_CODE_NO : WORD ;
    RBT19_WELD_COUNT : WORD ;
    RBT20_BT_CODE_NO : WORD ;
    RBT20_WELD_COUNT : WORD ;
    RBT21_BT_CODE_NO : WORD ;
    RBT21_WELD_COUNT : WORD ;
    RBT22_BT_CODE_NO : WORD ;
    RBT22_WELD_COUNT : WORD ;
    RBT23_BT_CODE_NO : WORD ;
    RBT23_WELD_COUNT : WORD ;
    RBT24_BT_CODE_NO : WORD ;
    RBT24_WELD_COUNT : WORD ;
    WELD_DETERMINES_RESULT : WORD ;
    WELD_CHECK_SUM : WORD ;
    SPARE1 : WORD ;
   END_STRUCT ;
   S711_WELD_BUFF_DATA61 : STRUCT
    STATION_MAIN : WORD ;
    DISTINCTION_LH_RH : WORD ;
    STAION_NUMBER : WORD ;
    VIN_NUMBER1 : WORD ;
    VIN_NUMBER2 : WORD ;
    VIN_NUMBER3 : WORD ;
    VIN_NUMBER4 : WORD ;
    SEQ_NUMBER1 : WORD ;
    SEQ_NUMBER2 : WORD ;
    RBT1_BT_CODE_NO : WORD ;
    RBT1_WELD_COUNT : WORD ;
    RBT2_BT_CODE_NO : WORD ;
    RBT2_WELD_COUNT : WORD ;
    RBT3_BT_CODE_NO : WORD ;
    RBT3_WELD_COUNT : WORD ;
    RBT4_BT_CODE_NO : WORD ;
    RBT4_WELD_COUNT : WORD ;
    RBT5_BT_CODE_NO : WORD ;
    RBT5_WELD_COUNT : WORD ;
    RBT6_BT_CODE_NO : WORD ;
    RBT6_WELD_COUNT : WORD ;
    RBT7_BT_CODE_NO : WORD ;
    RBT7_WELD_COUNT : WORD ;
    RBT8_BT_CODE_NO : WORD ;
    RBT8_WELD_COUNT : WORD ;
    RBT9_BT_CODE_NO : WORD ;
    RBT9_WELD_COUNT : WORD ;
    RBT10_BT_CODE_NO : WORD ;
    RBT10_WELD_COUNT : WORD ;
    RBT11_BT_CODE_NO : WORD ;
    RBT11_WELD_COUNT : WORD ;
    RBT12_BT_CODE_NO : WORD ;
    RBT12_WELD_COUNT : WORD ;
    RBT13_BT_CODE_NO : WORD ;
    RBT13_WELD_COUNT : WORD ;
    RBT14_BT_CODE_NO : WORD ;
    RBT14_WELD_COUNT : WORD ;
    RBT15_BT_CODE_NO : WORD ;
    RBT15_WELD_COUNT : WORD ;
    RBT16_BT_CODE_NO : WORD ;
    RBT16_WELD_COUNT : WORD ;
    RBT17_BT_CODE_NO : WORD ;
    RBT17_WELD_COUNT : WORD ;
    RBT18_BT_CODE_NO : WORD ;
    RBT18_WELD_COUNT : WORD ;
    RBT19_BT_CODE_NO : WORD ;
    RBT19_WELD_COUNT : WORD ;
    RBT20_BT_CODE_NO : WORD ;
    RBT20_WELD_COUNT : WORD ;
    RBT21_BT_CODE_NO : WORD ;
    RBT21_WELD_COUNT : WORD ;
    RBT22_BT_CODE_NO : WORD ;
    RBT22_WELD_COUNT : WORD ;
    RBT23_BT_CODE_NO : WORD ;
    RBT23_WELD_COUNT : WORD ;
    RBT24_BT_CODE_NO : WORD ;
    RBT24_WELD_COUNT : WORD ;
    WELD_DETERMINES_RESULT : WORD ;
    WELD_CHECK_SUM : WORD ;
    SPARE1 : WORD ;
   END_STRUCT ;
   S711_WELD_BUFF_DATA71 : STRUCT
    STATION_MAIN : WORD ;
    DISTINCTION_LH_RH : WORD ;
    STAION_NUMBER : WORD ;
    VIN_NUMBER1 : WORD ;
    VIN_NUMBER2 : WORD ;
    VIN_NUMBER3 : WORD ;
    VIN_NUMBER4 : WORD ;
    SEQ_NUMBER1 : WORD ;
    SEQ_NUMBER2 : WORD ;
    RBT1_BT_CODE_NO : WORD ;
    RBT1_WELD_COUNT : WORD ;
    RBT2_BT_CODE_NO : WORD ;
    RBT2_WELD_COUNT : WORD ;
    RBT3_BT_CODE_NO : WORD ;
    RBT3_WELD_COUNT : WORD ;
    RBT4_BT_CODE_NO : WORD ;
    RBT4_WELD_COUNT : WORD ;
    RBT5_BT_CODE_NO : WORD ;
    RBT5_WELD_COUNT : WORD ;
    RBT6_BT_CODE_NO : WORD ;
    RBT6_WELD_COUNT : WORD ;
    RBT7_BT_CODE_NO : WORD ;
    RBT7_WELD_COUNT : WORD ;
    RBT8_BT_CODE_NO : WORD ;
    RBT8_WELD_COUNT : WORD ;
    RBT9_BT_CODE_NO : WORD ;
    RBT9_WELD_COUNT : WORD ;
    RBT10_BT_CODE_NO : WORD ;
    RBT10_WELD_COUNT : WORD ;
    RBT11_BT_CODE_NO : WORD ;
    RBT11_WELD_COUNT : WORD ;
    RBT12_BT_CODE_NO : WORD ;
    RBT12_WELD_COUNT : WORD ;
    RBT13_BT_CODE_NO : WORD ;
    RBT13_WELD_COUNT : WORD ;
    RBT14_BT_CODE_NO : WORD ;
    RBT14_WELD_COUNT : WORD ;
    RBT15_BT_CODE_NO : WORD ;
    RBT15_WELD_COUNT : WORD ;
    RBT16_BT_CODE_NO : WORD ;
    RBT16_WELD_COUNT : WORD ;
    RBT17_BT_CODE_NO : WORD ;
    RBT17_WELD_COUNT : WORD ;
    RBT18_BT_CODE_NO : WORD ;
    RBT18_WELD_COUNT : WORD ;
    RBT19_BT_CODE_NO : WORD ;
    RBT19_WELD_COUNT : WORD ;
    RBT20_BT_CODE_NO : WORD ;
    RBT20_WELD_COUNT : WORD ;
    RBT21_BT_CODE_NO : WORD ;
    RBT21_WELD_COUNT : WORD ;
    RBT22_BT_CODE_NO : WORD ;
    RBT22_WELD_COUNT : WORD ;
    RBT23_BT_CODE_NO : WORD ;
    RBT23_WELD_COUNT : WORD ;
    RBT24_BT_CODE_NO : WORD ;
    RBT24_WELD_COUNT : WORD ;
    WELD_DETERMINES_RESULT : WORD ;
    WELD_CHECK_SUM : WORD ;
    SPARE1 : WORD ;
   END_STRUCT ;
   S711_WELD_BUFF_DATA81 : STRUCT
    STATION_MAIN : WORD ;
    DISTINCTION_LH_RH : WORD ;
    STAION_NUMBER : WORD ;
    VIN_NUMBER1 : WORD ;
    VIN_NUMBER2 : WORD ;
    VIN_NUMBER3 : WORD ;
    VIN_NUMBER4 : WORD ;
    SEQ_NUMBER1 : WORD ;
    SEQ_NUMBER2 : WORD ;
    RBT1_BT_CODE_NO : WORD ;
    RBT1_WELD_COUNT : WORD ;
    RBT2_BT_CODE_NO : WORD ;
    RBT2_WELD_COUNT : WORD ;
    RBT3_BT_CODE_NO : WORD ;
    RBT3_WELD_COUNT : WORD ;
    RBT4_BT_CODE_NO : WORD ;
    RBT4_WELD_COUNT : WORD ;
    RBT5_BT_CODE_NO : WORD ;
    RBT5_WELD_COUNT : WORD ;
    RBT6_BT_CODE_NO : WORD ;
    RBT6_WELD_COUNT : WORD ;
    RBT7_BT_CODE_NO : WORD ;
    RBT7_WELD_COUNT : WORD ;
    RBT8_BT_CODE_NO : WORD ;
    RBT8_WELD_COUNT : WORD ;
    RBT9_BT_CODE_NO : WORD ;
    RBT9_WELD_COUNT : WORD ;
    RBT10_BT_CODE_NO : WORD ;
    RBT10_WELD_COUNT : WORD ;
    RBT11_BT_CODE_NO : WORD ;
    RBT11_WELD_COUNT : WORD ;
    RBT12_BT_CODE_NO : WORD ;
    RBT12_WELD_COUNT : WORD ;
    RBT13_BT_CODE_NO : WORD ;
    RBT13_WELD_COUNT : WORD ;
    RBT14_BT_CODE_NO : WORD ;
    RBT14_WELD_COUNT : WORD ;
    RBT15_BT_CODE_NO : WORD ;
    RBT15_WELD_COUNT : WORD ;
    RBT16_BT_CODE_NO : WORD ;
    RBT16_WELD_COUNT : WORD ;
    RBT17_BT_CODE_NO : WORD ;
    RBT17_WELD_COUNT : WORD ;
    RBT18_BT_CODE_NO : WORD ;
    RBT18_WELD_COUNT : WORD ;
    RBT19_BT_CODE_NO : WORD ;
    RBT19_WELD_COUNT : WORD ;
    RBT20_BT_CODE_NO : WORD ;
    RBT20_WELD_COUNT : WORD ;
    RBT21_BT_CODE_NO : WORD ;
    RBT21_WELD_COUNT : WORD ;
    RBT22_BT_CODE_NO : WORD ;
    RBT22_WELD_COUNT : WORD ;
    RBT23_BT_CODE_NO : WORD ;
    RBT23_WELD_COUNT : WORD ;
    RBT24_BT_CODE_NO : WORD ;
    RBT24_WELD_COUNT : WORD ;
    WELD_DETERMINES_RESULT : WORD ;
    WELD_CHECK_SUM : WORD ;
    SPARE1 : WORD ;
   END_STRUCT ;
   S711_WELD_BUFF_DATA91 : STRUCT
    STATION_MAIN : WORD ;
    DISTINCTION_LH_RH : WORD ;
    STAION_NUMBER : WORD ;
    VIN_NUMBER1 : WORD ;
    VIN_NUMBER2 : WORD ;
    VIN_NUMBER3 : WORD ;
    VIN_NUMBER4 : WORD ;
    SEQ_NUMBER1 : WORD ;
    SEQ_NUMBER2 : WORD ;
    RBT1_BT_CODE_NO : WORD ;
    RBT1_WELD_COUNT : WORD ;
    RBT2_BT_CODE_NO : WORD ;
    RBT2_WELD_COUNT : WORD ;
    RBT3_BT_CODE_NO : WORD ;
    RBT3_WELD_COUNT : WORD ;
    RBT4_BT_CODE_NO : WORD ;
    RBT4_WELD_COUNT : WORD ;
    RBT5_BT_CODE_NO : WORD ;
    RBT5_WELD_COUNT : WORD ;
    RBT6_BT_CODE_NO : WORD ;
    RBT6_WELD_COUNT : WORD ;
    RBT7_BT_CODE_NO : WORD ;
    RBT7_WELD_COUNT : WORD ;
    RBT8_BT_CODE_NO : WORD ;
    RBT8_WELD_COUNT : WORD ;
    RBT9_BT_CODE_NO : WORD ;
    RBT9_WELD_COUNT : WORD ;
    RBT10_BT_CODE_NO : WORD ;
    RBT10_WELD_COUNT : WORD ;
    RBT11_BT_CODE_NO : WORD ;
    RBT11_WELD_COUNT : WORD ;
    RBT12_BT_CODE_NO : WORD ;
    RBT12_WELD_COUNT : WORD ;
    RBT13_BT_CODE_NO : WORD ;
    RBT13_WELD_COUNT : WORD ;
    RBT14_BT_CODE_NO : WORD ;
    RBT14_WELD_COUNT : WORD ;
    RBT15_BT_CODE_NO : WORD ;
    RBT15_WELD_COUNT : WORD ;
    RBT16_BT_CODE_NO : WORD ;
    RBT16_WELD_COUNT : WORD ;
    RBT17_BT_CODE_NO : WORD ;
    RBT17_WELD_COUNT : WORD ;
    RBT18_BT_CODE_NO : WORD ;
    RBT18_WELD_COUNT : WORD ;
    RBT19_BT_CODE_NO : WORD ;
    RBT19_WELD_COUNT : WORD ;
    RBT20_BT_CODE_NO : WORD ;
    RBT20_WELD_COUNT : WORD ;
    RBT21_BT_CODE_NO : WORD ;
    RBT21_WELD_COUNT : WORD ;
    RBT22_BT_CODE_NO : WORD ;
    RBT22_WELD_COUNT : WORD ;
    RBT23_BT_CODE_NO : WORD ;
    RBT23_WELD_COUNT : WORD ;
    RBT24_BT_CODE_NO : WORD ;
    RBT24_WELD_COUNT : WORD ;
    WELD_DETERMINES_RESULT : WORD ;
    WELD_CHECK_SUM : WORD ;
    SPARE1 : WORD ;
   END_STRUCT ;
   S711_WELD_BUFF_DATA101 : STRUCT
    STATION_MAIN : WORD ;
    DISTINCTION_LH_RH : WORD ;
    STAION_NUMBER : WORD ;
    VIN_NUMBER1 : WORD ;
    VIN_NUMBER2 : WORD ;
    VIN_NUMBER3 : WORD ;
    VIN_NUMBER4 : WORD ;
    SEQ_NUMBER1 : WORD ;
    SEQ_NUMBER2 : WORD ;
    RBT1_BT_CODE_NO : WORD ;
    RBT1_WELD_COUNT : WORD ;
    RBT2_BT_CODE_NO : WORD ;
    RBT2_WELD_COUNT : WORD ;
    RBT3_BT_CODE_NO : WORD ;
    RBT3_WELD_COUNT : WORD ;
    RBT4_BT_CODE_NO : WORD ;
    RBT4_WELD_COUNT : WORD ;
    RBT5_BT_CODE_NO : WORD ;
    RBT5_WELD_COUNT : WORD ;
    RBT6_BT_CODE_NO : WORD ;
    RBT6_WELD_COUNT : WORD ;
    RBT7_BT_CODE_NO : WORD ;
    RBT7_WELD_COUNT : WORD ;
    RBT8_BT_CODE_NO : WORD ;
    RBT8_WELD_COUNT : WORD ;
    RBT9_BT_CODE_NO : WORD ;
    RBT9_WELD_COUNT : WORD ;
    RBT10_BT_CODE_NO : WORD ;
    RBT10_WELD_COUNT : WORD ;
    RBT11_BT_CODE_NO : WORD ;
    RBT11_WELD_COUNT : WORD ;
    RBT12_BT_CODE_NO : WORD ;
    RBT12_WELD_COUNT : WORD ;
    RBT13_BT_CODE_NO : WORD ;
    RBT13_WELD_COUNT : WORD ;
    RBT14_BT_CODE_NO : WORD ;
    RBT14_WELD_COUNT : WORD ;
    RBT15_BT_CODE_NO : WORD ;
    RBT15_WELD_COUNT : WORD ;
    RBT16_BT_CODE_NO : WORD ;
    RBT16_WELD_COUNT : WORD ;
    RBT17_BT_CODE_NO : WORD ;
    RBT17_WELD_COUNT : WORD ;
    RBT18_BT_CODE_NO : WORD ;
    RBT18_WELD_COUNT : WORD ;
    RBT19_BT_CODE_NO : WORD ;
    RBT19_WELD_COUNT : WORD ;
    RBT20_BT_CODE_NO : WORD ;
    RBT20_WELD_COUNT : WORD ;
    RBT21_BT_CODE_NO : WORD ;
    RBT21_WELD_COUNT : WORD ;
    RBT22_BT_CODE_NO : WORD ;
    RBT22_WELD_COUNT : WORD ;
    RBT23_BT_CODE_NO : WORD ;
    RBT23_WELD_COUNT : WORD ;
    RBT24_BT_CODE_NO : WORD ;
    RBT24_WELD_COUNT : WORD ;
    WELD_DETERMINES_RESULT : WORD ;
    WELD_CHECK_SUM : WORD ;
    SPARE1 : WORD ;
   END_STRUCT ;
  END_STRUCT ;
BEGIN
   S711A_WELD_BUFF_DATA1.STATION_MAIN := W#16#0;
   S711A_WELD_BUFF_DATA1.DISTINCTION_LH_RH := W#16#0;
   S711A_WELD_BUFF_DATA1.STAION_NUMBER := W#16#0;
   S711A_WELD_BUFF_DATA1.VIN_NUMBER1 := W#16#0;
   S711A_WELD_BUFF_DATA1.VIN_NUMBER2 := W#16#0;
   S711A_WELD_BUFF_DATA1.VIN_NUMBER3 := W#16#0;
   S711A_WELD_BUFF_DATA1.VIN_NUMBER4 := W#16#0;
   S711A_WELD_BUFF_DATA1.SEQ_NUMBER1 := W#16#0;
   S711A_WELD_BUFF_DATA1.SEQ_NUMBER2 := W#16#0;
   S711A_WELD_BUFF_DATA1.RBT1_BT_CODE_NO := W#16#0;
   S711A_WELD_BUFF_DATA1.RBT1_WELD_COUNT := W#16#0;
   S711A_WELD_BUFF_DATA1.RBT2_BT_CODE_NO := W#16#0;
   S711A_WELD_BUFF_DATA1.RBT2_WELD_COUNT := W#16#0;
   S711A_WELD_BUFF_DATA1.RBT3_BT_CODE_NO := W#16#0;
   S711A_WELD_BUFF_DATA1.RBT3_WELD_COUNT := W#16#0;
   S711A_WELD_BUFF_DATA1.RBT4_BT_CODE_NO := W#16#0;
   S711A_WELD_BUFF_DATA1.RBT4_WELD_COUNT := W#16#0;
   S711A_WELD_BUFF_DATA1.RBT5_BT_CODE_NO := W#16#0;
   S711A_WELD_BUFF_DATA1.RBT5_WELD_COUNT := W#16#0;
   S711A_WELD_BUFF_DATA1.RBT6_BT_CODE_NO := W#16#0;
   S711A_WELD_BUFF_DATA1.RBT6_WELD_COUNT := W#16#0;
   S711A_WELD_BUFF_DATA1.RBT7_BT_CODE_NO := W#16#0;
   S711A_WELD_BUFF_DATA1.RBT7_WELD_COUNT := W#16#0;
   S711A_WELD_BUFF_DATA1.RBT8_BT_CODE_NO := W#16#0;
   S711A_WELD_BUFF_DATA1.RBT8_WELD_COUNT := W#16#0;
   S711A_WELD_BUFF_DATA1.RBT9_BT_CODE_NO := W#16#0;
   S711A_WELD_BUFF_DATA1.RBT9_WELD_COUNT := W#16#0;
   S711A_WELD_BUFF_DATA1.RBT10_BT_CODE_NO := W#16#0;
   S711A_WELD_BUFF_DATA1.RBT10_WELD_COUNT := W#16#0;
   S711A_WELD_BUFF_DATA1.RBT11_BT_CODE_NO := W#16#0;
   S711A_WELD_BUFF_DATA1.RBT11_WELD_COUNT := W#16#0;
   S711A_WELD_BUFF_DATA1.RBT12_BT_CODE_NO := W#16#0;
   S711A_WELD_BUFF_DATA1.RBT12_WELD_COUNT := W#16#0;
